	fbAchse_Buerste_030801.IsReset:= P_ServiceAchsen.xStopAktiv_Reset[AxId_Buerste_030801];
	fbAchse_Buerste_030801.IsFreigabe:= P_ServiceAchsen.xFreigabe_Aktiv[AxId_Buerste_030801];
	fbAchse_Buerste_030801.IwZielSollwert:= P_ServiceAchsen.rZielSollwert[AxId_Buerste_030801];
	fbAchse_Buerste_030801.IwSpeed:= P_ServiceAchsen.uiSpeed[AxId_Buerste_030801];
ELSE
	IF	fbEins[iEins_Id].OsAutomatikEin
		OR	fbEins[iEins_Id].OsHandEin
			AND	astrGButtonManTransporte[ID_Buerste_030801_Positionieren].bSchalt
	THEN
		arGZielAchse[AxId_Buerste_030801]:= st_Achse_Buerste_030801.rZiel;
		arGSpeedAchse[AxId_Buerste_030801]:= st_Achse_Buerste_030801.rSpeed;
		abGStartAchse[AxId_Buerste_030801]:= st_Achse_Buerste_030801.xStartPosi;
		abGEichenAchse[AxId_Buerste_030801]:= st_Achse_Buerste_030801.xStartEichen;
		abGFreigabeAchse[AxId_Buerste_030801]:= st_Achse_Buerste_030801.xFreigabe;
	ELSE
		abGStartAchse[AxId_Buerste_030801]:= FALSE;
		abGEichenAchse[AxId_Buerste_030801]:= FALSE;
		abGFreigabeAchse[AxId_Buerste_030801]:= FALSE;
	END_IF;

	fbAchse_Buerste_030801.IsReset:=
		( astrGButtonManTransporte[ID_Buerste_030801_Tippen].bSchalt
			OR	astrGButtonManTransporte[ID_Buerste_030801_Positionieren].bSchalt )
		AND 	strGLmHand.bI_Reset
		OR NOT fbEins[iEins_Id].OsAutomatikEin
			AND	GDat.TrE_Daten[TrEId_030801_Buerste].iReset <> 0;

	fbAchse_Buerste_030801.IsFreigabe:=
		( abGFreigabeAchse[AxId_Buerste_030801]
			AND NOT bFehlerFahrenFreigabe_Buerste_030801
			AND NOT bFehlerFahrenPlus_Buerste_030801
			AND NOT bFehlerFahrenMinus_Buerste_030801
			OR NOT fbAchse_Buerste_030801.IsAutomatik
				AND	fbAchse_Buerste_030801.IsHand )
		AND	fbEins[iEins_Id].OsNotHaltIstOk
		AND NOT fbAchse_Buerste_030801.OwOut.xAchseFehler
		AND	gxAlleTuerenGeschlossen_HardwareC[giSicher_C2_2]
		AND	gxAlleTuerenGeschlossenVerriegelt_HardwareC[giSicher_C2_2]
		AND	gxAlleTuerenGeschlossen_FreigabeAchseC[giSicher_C2_2];

	IF	fbEins[iEins_Id].OsAutomatikEin
		AND	arGSpeedAchse[AxId_Buerste_030801] > 0
	THEN
		fbAchse_Buerste_030801.IwSpeed:=
			LIMIT ( 0.1,arGSpeedAchse[AxId_Buerste_030801],100 );
	ELSE
		fbAchse_Buerste_030801.IwSpeed:= 100;
	END_IF;

	IF	fbAchse_Buerste_030801.IsSichereGeschwindigkeit
	THEN
		fbAchse_Buerste_030801.IwSpeed_HandSlow:= 50;
		fbAchse_Buerste_030801.IwSpeed_HandFast:= 100;
	ELSE
		fbAchse_Buerste_030801.IwSpeed_HandSlow:= 50;
		fbAchse_Buerste_030801.IwSpeed_HandFast:= 100;
	END_IF;

	fbAchse_Buerste_030801.IwBeschleunigung:= st_Achse_Buerste_030801.rBeschleunigung;
	fbAchse_Buerste_030801.IwVerzoegerung:= st_Achse_Buerste_030801.rVerzoegerung;
	fbAchse_Buerste_030801.IwRuck:= st_Achse_Buerste_030801.rRuck;

	fbAchse_Buerste_030801.IsStartEichen:=
		abGEichenAchse[AxId_Buerste_030801]
		AND NOT gxTestbetriebOhneMaschineAktiv;

	fbAchse_Buerste_030801.IwZielSollwert:=
		arGZielAchse[AxId_Buerste_030801];

	fbAchse_Buerste_030801.IsStartAufPosition:=
		abGStartAchse[AxId_Buerste_030801]
		AND 	fbAchse_Buerste_030801.IsFreigabe
		AND	fbAchse_Buerste_030801.OwOut.xAchseGeeicht;

	fbAchse_Buerste_030801.IsNeueGeschwindigkeit:= st_Achse_Buerste_030801.xStartNeueGeschwindigkeit;

	fbAchse_Buerste_030801.IsSonderGeschwindigkeit:= st_Achse_Buerste_030801.xSonderGeschwindigkeit;
	fbAchse_Buerste_030801.IwSonderGeschwindigkeit:= LREAL_TO_REAL ( st_Achse_Buerste_030801.lrSonderGeschwindigkeit );

	fbAchse_Buerste_030801.IsStartNeuesZielWaehrendPosi:= st_Achse_Buerste_030801.xStartNeuesZielWaehrendPosi;
	fbAchse_Buerste_030801.IwNeuesZielWaehrendPosi:= st_Achse_Buerste_030801.rNeuesZielWaehrendPosi;

	IF	fbAchse_Buerste_030801.xZielUmschiessen
	THEN
		st_Achse_Buerste_030801.xStartNeuesZielWaehrendPosi:= FALSE;
	END_IF;

	IF	fbAchse_Buerste_030801.xGeschwindigkeitUmschiessen
	THEN
		st_Achse_Buerste_030801.xStartNeueGeschwindigkeit:= FALSE;
	END_IF;
END_IF;

fbAchse_Buerste_030801();

IF	fbAchse_Buerste_030801.IsHand
	AND	fbAchse_Buerste_030801.IsReset
	OR NOT bAchseBeiStartGeeicht_Buerste_030801
THEN
	abGAchseNeuEichen[AxId_Buerste_030801]:= TRUE;
	bAchseBeiStartGeeicht_Buerste_030801:= TRUE;
END_IF;

(*------------------------------------------------------*)
(*  Handling: -> Jobverteiler                      	  *)
(*------------------------------------------------------*)

st_Achse_Buerste_030801.iID:= AxId_Buerste_030801;
st_Achse_Buerste_030801.xNichtEichen:= TRUE;
st_Achse_Buerste_030801.stVonAchse:= fbAchse_Buerste_030801.OwOut;
st_Achse_Buerste_030801.stVonAchse.xAchseGeeicht:=
	fbAchse_Buerste_030801.OwOut.xAchseGeeicht;

st_Achse_Buerste_030801.xBereit_FuerFahrjob:=
	fbAchse_Buerste_030801.OwOut.xAchseBereit
	AND NOT fbAchse_Buerste_030801.OwOut.xAchseFehler;



(*-----------------------------------------------------------------*)
(* Die globale Struktur für die Leuchtmelde Handtasten beschreiben *)
(*-----------------------------------------------------------------*)
IF	fbAchse_Buerste_030801.IsHand
	AND	astrGButtonManTransporte[ID_Buerste_030801_Tippen].bSchalt
THEN
	IF NOT fbAchse_Buerste_030801.IsEsEndlagePlus
	THEN
		strGLmHand.bQ_Heben:= TRUE;
	END_IF;

	IF NOT fbAchse_Buerste_030801.IsEsEndlageMinus
	THEN
		strGLmHand.bQ_Senken:= TRUE;
	END_IF;
END_IF;



				(*---------------------------------------------------*)
				(*---------------------------------------------------*)
				(*           Freigabe Hardwaren / Software           *)
				(*---------------------------------------------------*)
				(*---------------------------------------------------*)

abGAchseDisable[AxId_Buerste_030801]:=
	GKoAnB[usiBuerste1].xInAktiv;

IF ( fbAchse_Buerste_030801.IsEsEndlageMinus
		OR 	fbAchse_Buerste_030801.IsEsEndlagePlus )
	AND NOT gxTestbetriebOhneMaschineAktiv
THEN
	abGEndlageAngefahren[AxId_Buerste_030801]:= TRUE;
END_IF;

IF	strGLmHand.bI_QuittStoerung
		AND NOT fbAchse_Buerste_030801.IsEsEndlageMinus
		AND NOT fbAchse_Buerste_030801.IsEsEndlagePlus
	OR NOT fbEins[iEins_Id].OsSteuerspannungIstEin
THEN
	abGEndlageFreifahren[AxId_Buerste_030801]:= FALSE;
	abGEndlageAngefahren[AxId_Buerste_030801]:= FALSE;
END_IF;

abGEndlageFreifahren[AxId_Buerste_030801]:=
	fbEins[iEins_Id].OsHandEin
	AND	abGEndlageAngefahren[AxId_Buerste_030801];

aTonGReglerfreigabe[AxId_Buerste_030801].IN:=
	( NOT abGEndlageAngefahren[AxId_Buerste_030801]
		OR	abGEndlageFreifahren[AxId_Buerste_030801] )
	AND	bFreigabeFahren_Buerste_030801
	AND NOT abGAchseDisable[AxId_Buerste_030801]
	AND NOT AxFrNcFehler[AxId_Buerste_030801]
	AND NOT fbAchse_Buerste_030801.OsMFehlerMcBausteine
	AND NOT GKoAnB[usiBuerste1].xInAktiv;

aTonGReglerfreigabe[AxId_Buerste_030801](PT:= T#500MS);

abGReglerfreigabe[AxId_Buerste_030801]:=
	aTonGReglerfreigabe[AxId_Buerste_030801].Q
	OR	aTofGReglerfreigabe_Aus[AxId_Buerste_030801].Q
		AND	AxFrNcFahrePlus[AxId_Buerste_030801]
		AND NOT abGEndlageAngefahren[AxId_Buerste_030801]
	OR	aTofGReglerfreigabe_Aus[AxId_Buerste_030801].Q
		AND	AxFrNcFahreMinus[AxId_Buerste_030801]
		AND NOT abGEndlageAngefahren[AxId_Buerste_030801];

(* Ausschaltverzoegerung Reglerfreigabe *)
aTofGReglerfreigabe_Aus[AxId_Buerste_030801].IN:=
	aTonGReglerfreigabe[AxId_Buerste_030801].IN
		AND  	aTonGReglerfreigabe[AxId_Buerste_030801].Q;
aTofGReglerfreigabe_Aus[AxId_Buerste_030801](PT:= GKoAll.tBisReglerfreigabeAus_BeiNotHalt);

aTonGVorschubfreigabe[AxId_Buerste_030801](PT:= T#500MS);

aTonGVorschubfreigabe[AxId_Buerste_030801].IN:=
	abGReglerfreigabe[AxId_Buerste_030801];

abGVorschubfreigabe[AxId_Buerste_030801]:= aTonGVorschubfreigabe[AxId_Buerste_030801].Q;

abGVorschubfreigabePlus[AxId_Buerste_030801]:=
	NOT fbAchse_Buerste_030801.IsEsEndlagePlus
	OR	gxTestbetriebOhneMaschineAktiv;

abGVorschubfreigabeMinus[AxId_Buerste_030801]:=
	NOT fbAchse_Buerste_030801.IsEsEndlageMinus
	OR	gxTestbetriebOhneMaschineAktiv;

(*---------------------------------------------------*)
(* Achse: Freigabe Software              		     *)
(*---------------------------------------------------*)

AxToNcRfg[AxId_Buerste_030801]:=
	abGReglerfreigabe[AxId_Buerste_030801]
		AND NOT abGAchseDisable[AxId_Buerste_030801];

AxToNcVfp[AxId_Buerste_030801]:=
	abGVorschubfreigabe[AxId_Buerste_030801]
		AND	abGVorschubfreigabePlus[AxId_Buerste_030801]
		AND	aTonGReglerfreigabe[AxId_Buerste_030801].Q
		AND NOT abGAchseDisable[AxId_Buerste_030801];

AxToNcVfm[AxId_Buerste_030801]:=
	abGVorschubfreigabe[AxId_Buerste_030801]
		AND	abGVorschubfreigabeMinus[AxId_Buerste_030801]
		AND	aTonGReglerfreigabe[AxId_Buerste_030801].Q
		AND NOT abGAchseDisable[AxId_Buerste_030801];

(*---------------------------------------------------*)
(* Achse: Ausgänge an Systemmanager schreiben	     *)
(*---------------------------------------------------*)
bQW10SchwertbObZMinus		:= bIW10DirectionMinus;
bQW10SchwertbObZPlus		:= bIW10DirectionPlus;
bQW10SchwertbObZSchnell		:= bIW10VeloHigh;
END_ACTION

ACTION Up_15_EilSchl_PosiBuerste_030801:
(*------------------------------------------------*)
(*------------------------------------------------*)
(* Achse: Jobhandling Positionierung		  *)
(*------------------------------------------------*)
(*------------------------------------------------*)
(*
IF GDat.TrE_Daten[TrEId_030801].iAnzahlPlatten > 0
THEN
	bKleinteilBuerste_030801:= FALSE;

	FOR i:= 1 TO LIMIT(1,GDat.TrE_Daten[TrEId_030801].iAnzahlPlatten,giMaxAnzahlPlattenProSpur)
	DO
		IF	(GDat.TrE_Daten[TrEId_030801].arLaenge[i] <= GKoAnB[usiBuerste1].rMinLaenge_Buerste
				OR GDat.TrE_Daten[TrEId_030801].arBreite[i] <= GKoAnB[usiBuerste1].rMinBreite_Buerste)
		THEN
			bKleinteilBuerste_030801:= TRUE;
			EXIT;
		END_IF;
	END_FOR;

	rDickeBuerste	:= GDat.TrE_Daten[TrEId_030801].arDicke[1];
	rBreiteBuerste	:= GDat.TrE_Daten[TrEId_030801].arBreite[1];

ELSIF ( GDat.TrE_Daten[TrEId_030801].iJobStatus = iDatenAktiv
		OR GDat.TrE_Daten[TrEId_030801].iJobStatus = iUebernahmeGestartet )
	AND GDat.TrE_Daten[TrEId_030801].iAnzahlPlatten = 0
THEN
	bKleinteilBuerste_030801:= FALSE;

	FOR i:= 1 TO LIMIT(1,fbJobBahn030801.strBahnjob_Aktiv.iAnzahlPlatten,giMaxAnzahlPlattenProSpur)
	DO
		IF	(fbJobBahn030801.strBahnjob_Aktiv.arLaenge[i] <= GKoAnB[usiBuerste1].rMinLaenge_Buerste
				OR fbJobBahn030801.strBahnjob_Aktiv.arBreite[i] <= GKoAnB[usiBuerste1].rMinBreite_Buerste)
		THEN
			bKleinteilBuerste_030801:= TRUE;
			EXIT;
		END_IF;
	END_FOR;

	rDickeBuerste	:= fbJobBahn030801.strBahnjob_Aktiv.arDicke[1];
	rBreiteBuerste	:= fbJobBahn030801.strBahnjob_Aktiv.arBreite[1];

ELSIF GDat.TrE_Daten[TrEId_030801].iJobStatus = iSekNichtAktiv
	AND GDat.TrE_Daten[TrEId_030801].iAnzahlPlatten = 0
	AND GDat.TrE_Daten[TrEId_070402].iAnzahlPlatten > 0
THEN

	bKleinteilBuerste_030801:= FALSE;

	FOR i:= 1 TO LIMIT(1,GDat.TrE_Daten[TrEId_070402].iAnzahlPlatten,giMaxAnzahlPlattenProSpur)
	DO
		IF	(GDat.TrE_Daten[TrEId_070402].arLaenge[i] <= GKoAnB[usiBuerste1].rMinLaenge_Buerste
				OR GDat.TrE_Daten[TrEId_070402].arBreite[i] <= GKoAnB[usiBuerste1].rMinBreite_Buerste)
		THEN
			bKleinteilBuerste_030801:= TRUE;
			EXIT;
		END_IF;
	END_FOR;

	rDickeBuerste	:= GDat.TrE_Daten[TrEId_070402].arDicke[1];
	rBreiteBuerste	:= GDat.TrE_Daten[TrEId_070402].arBreite[1];

ELSIF GDat.TrE_Daten[TrEId_030801].iAnzahlPlatten = 0
	AND	GDat.TrE_Daten[TrEId_030801].asBarcode[1] = ''
	AND 	strGHdshk_Bahn030801.str_BahnStatus = iAutomatikBereitJob
	AND NOT strGHdshk_Bahn030801.b_BahnBelegt
THEN
	bKleinteilBuerste_030801:= FALSE;
END_IF;

fbTOF_BuersteAntriebEin_030801(
		IN:= strGHdshk_Bahn030801.b_BahnVor,
		PT:= t#5s,
		Q=> ,
		ET=> );

fbEntprellenHoehenkontrolle_030801(
	IsSensor:= NOT bIW308Hoehenkontr
					AND FALSE,
	tEntprell_Belegt:= t#1s,
	tEntprell_Frei:= t#1s,
	OsSensor=> );

IF	fbEntprellenHoehenkontrolle_030801.OsSensor
	AND NOT gxTestbetriebOhneMaschineAktiv
THEN
	bQ_MFehlerHoehenkontrolle030801:= TRUE;

ELSIF	bQ_MFehlerHoehenkontrolle030801
	AND (strGLmHand.bI_QuittStoerung
		OR (NOT fbEntprellenHoehenkontrolle_030801.OsSensor
			AND AxFrNc_fPosIst[AxId_Buerste_030801] >= (GDat.TrE_Daten[TrEId_030801].arDicke[1] - fbBuerste_030801.rToleranzBuerste)))
THEN
	bQ_MFehlerHoehenkontrolle030801:= FALSE;
END_IF
*)

fbBuerste_030801(
	sI_Name							:= '03.08.01_Buerste',
	uiI_AxId_Oben					:= AxId_Buerste_030801,
	uiI_ProId						:= P_BahnJob,
	bI_Hand							:= fbEins[iEins_Id].OsHandEin,
	bI_Automatik					:= fbEins[iEins_Id].OsAutomatikEin,
	bI_Reset						:= strGLmHand.bI_Reset
								 	 	AND ( astrGButtonManTransporte[ID_Buerste_030801_Tippen].bSchalt
									 		 OR	astrGButtonManTransporte[ID_Buerste_030801_Positionieren].bSchalt ),
	bI_QuittStoerung				:= strGLmHand.bI_QuittStoerung
										OR fbEins[iEins_Id].OsImpulsSteuerspannungEin,
	bI_ZyklusBeenden				:= fbEins[iEins_Id].OsZyklusBeenden
										OR	Aufruf_Allgemein.bAnforderungAnlageAus,
	bI_StoerungBuerstenAntriebOben	:= NOT bIW10SchwertbuersteObBtp,
	bI_StoerungBuerstenAntriebUnten	:= NOT bIW10SchwertbuersteUntBtp,
	bI_StoerungAchse				:= FALSE,
	bI_SicherheitOK					:= gxSicherheitsBereichQuittiertC[giSicher_C2_2],
	bI_Kleinteile					:= bKleinteilBuerste_030801,
	bI_BuersteZu					:= TRUE,
	bI_BuersteAntriebEin			:= strGHdshk_Bahn030801.b_BahnVor,
	bI_TeileBuersten				:= TRUE,
	bI_TeileReinigen				:= fbTOF_BuersteAntriebEin_030801.Q,
	bI_IngromatEin					:= FALSE,
	bI_FahrtInGrundOhneEichen		:= astrGButtonManTransporte[ID_Buerste_030801_Tippen].bSchalt
										OR	astrGButtonManTransporte[ID_Buerste_030801_Positionieren].bSchalt,
	bI_FreigabeAufPosition			:= fbBuerste_030801.rI_Dicke > 0,
	bI_EichenManuell				:= TRUE,
	bI_Testbetrieb					:= gxTestbetriebOhneMaschineAktiv,
	bI_ImpulsInit					:= bGImpulsInitSprache,
	rI_Dicke						:= fbJobBahn030801.strBahnjob_Aktiv.arDicke[1],
	rI_Breite						:= fbJobBahn030801.strBahnjob_Aktiv.arBreite[1], 
	strI_Para						:= GKoAnB[usiBuerste1],
	strIO_TrE_Extern 				:= GDat.TrE_Daten[TrEId_030801_Buerste],
	strIO_Hubachse_Oben				:= st_Achse_Buerste_030801,
	abQ_Blasventil					=> ,
	bQ_BuersteOeffnen				=> ,
	bQ_BuersteObenEin				=> bQW10SchwertbuersteObEin,
	bQ_BuersteUntenEin				=> bQW10SchwertbuersteUntEin,
	bQ_Reinigen						=> bQW10SchwertbReinigEin,
	bQ_Ingromat						=> ,
	bQ_ZyklusBeendet				=> ,
	bQ_Grundstellung				=> ,
	bQ_SchleichenEichenOben			=> ,
	bQ_IstwertSetzenOben=> ,
	bQ_MStoerungBuerstenAntriebOben=> ,
	bQ_MStoerungBuerstenAntriebUnten=> ,
	uiQ_Ablaufstatus=> , 
	strQ_Status=> );

	
IF	astrGButtonManTransporte[ID_Buerste_030801_Tippen].bSchalt
	OR	astrGButtonManTransporte[ID_Buerste_030801_Positionieren].bSchalt
THEN
	TZeile.Aktiv := TRUE;
	TZeile.Wert  := REAL_TO_INT(AxFrNc_fPosIst[AxId_Buerste_030801]);
END_IF;

IF	( fbBuerste_030801.strQ_Status = iAutomatikBereitJob
		AND	fbBuerste_030801.rI_Dicke > 0
		AND	st_Achse_Buerste_030801.xBereit_FuerFahrjob
		AND 	(( ABS (( fbBuerste_030801.rI_Dicke + fbBuerste_030801.strI_Para.rOeffnungswertKleinteile_Oben ) - fbBuerste_030801.rIstwert ) <= fbBuerste_030801.rToleranzBuerste
				AND	fbBuerste_030801.bI_Kleinteile )
			OR	( ABS ( fbBuerste_030801.rI_Dicke - fbBuerste_030801.rIstwert ) <= fbBuerste_030801.rToleranzBuerste
				AND NOT fbBuerste_030801.bI_Kleinteile )))
	OR	fbBuerste_030801.strI_Para.xInAktiv
THEN
	bBuersteInPostion_030801:= TRUE;
ELSE
	bBuersteInPostion_030801:= FALSE;
END_IF;
END_ACTION

ACTION Up_16_Anschlag_030201:

fbAnschlag_030201(
	IsHand									:= fbEins[iEins_Id].OsHandEin
												OR ( NOT fbEins[iEins_Id].OsAutomatikEin
													AND ( GDat.TrE_Daten[TrEId_030201_Roll1].iReset <> 0
														OR	GDat.TrE_Daten[TrEId_030202_Roll2].iReset <> 0 ) ),
	IsAutomatik								:= fbEins[iEins_Id].OsAutomatikEin,
	IsReset									:= astrGButtonManTransporte[ID_Anschlag030201].bSchalt
												AND	strGLmHand.bI_Reset
												OR ( NOT fbEins[iEins_Id].OsAutomatikEin
													AND ( GDat.TrE_Daten[TrEId_030201_Roll1].iReset <> 0
														OR GDat.TrE_Daten[TrEId_030202_Roll2].iReset <> 0 )),
	IsQuittStoerung							:= strGLmHand.bI_QuittStoerung,
	IsTestbetrieb							:= gxTestbetriebOhneMaschineAktiv,
	IsNotHaltIstOK							:= TRUE,
	IsFreigabe_Automatik					:= TRUE,
	IsStoerungAntrieb						:= strGStoerungen[iEins_Id].bStoerungDruckluft,
	IsSicherheitOK							:= gxSicherheitsBereichQuittiertC[giSicher_C2_1],
	IsTHandVor								:= astrGButtonManTransporte[ID_Anschlag030201].bSchalt
												AND	strGLmHand.bI_Senken,
	IsTHandZurueck							:= astrGButtonManTransporte[ID_Anschlag030201].bSchalt
												AND	strGLmHand.bI_Heben,
	IsDauerlauf_Aktivieren					:= astrGButtonManTransporte[ID_Anschlag030201].bSchalt
												AND	gxDauerlauf_Aktiv,
	IsHand_Takt								:= gTakt22,
	IsGrundstellung							:= bIW302Anschlag1Sek1GS
												AND NOT gxTestbetriebOhneMaschineAktiv
												OR	gxTestbetriebOhneMaschineAktiv
													AND	fbAnschlag_030201.OsGrundstellung,
	IsArbeitsstellung						:= bIW302Anschlag1Sek1AS
												AND NOT gxTestbetriebOhneMaschineAktiv
												OR	gxTestbetriebOhneMaschineAktiv
													AND	fbAnschlag_030201.OsArbeitsstellung,
	IwMode									:= 3,
	IwMode_NotHalt							:= 0,
	IwDoJob									:= strGHdshk_Anschlag030201.str_DoJob,
	IsFreigabeGrundposition					:= TRUE,
	IsGrundpositionArbeitsstellung			:= strGHdshk_Anschlag030201.b_Arbeitsstellung,
	IsKeineGrundposition					:= FALSE,
	IsOhneUeberwachung						:= FALSE,
	IsGesetzterOutMerken					:= TRUE,
	IsClearOut_NachJob						:= FALSE,
	IsOutAnlassen_Hand						:= TRUE,
	IsOutAnlassen_Stoerung					:= TRUE,
	IsPositionsUeberwachung					:= TRUE,
	IsBewegungsUeberwachung					:= TRUE,
	IwBisGrundstellung						:= strGHdshk_Anschlag030201.tBisGrundstellung,
	IwBisArbeitsstellung					:= strGHdshk_Anschlag030201.tBisArbeitsstellung,
	IwMaxLaufzeitZylinder					:= strGHdshk_Anschlag030201.tMaxLaufzeit,
	IwBisDrucklos							:= strGHdshk_Anschlag030201.tBisDrucklos,
	OsGrundstellung							=> bQW302AnschlagSek1GS,
	OsArbeitsstellung						=> bQW302AnschlagSek1AS,
	OwJobAktiv								=> strGHdshk_Anschlag030201.str_JobAktiv,
	OwStatus								=> strGHdshk_Anschlag030201.str_ZylinderStatus,
	OwAblaufStatus							=> strGHdshk_Anschlag030201.i_AblaufStatus,
	OsMStoerungAntrieb						=> strGHdshk_Anschlag030201.b_MStoerungAntrieb,
	OsMMaxLaufzeit_Ein						=> strGHdshk_Anschlag030201.b_MMaxLaufzeit_Ein,
	OsMMaxLaufzeit_Aus						=> strGHdshk_Anschlag030201.b_MMaxLaufzeit_Aus,
	OsMPositionsUeberwachung_Ein			=> strGHdshk_Anschlag030201.b_MPositionsUeberwachung_Ein,
	OsMPositionsUeberwachung_Aus			=> strGHdshk_Anschlag030201.b_MPositionsUeberwachung_Aus,
	OsMBewegungsUeberwachung				=> strGHdshk_Anschlag030201.b_MBewegungsUeberwachung);

	
strGHdshk_Anschlag030201.b_Arbeitsstellung:= fbAnschlag_030201.IsArbeitsstellung;
strGHdshk_Anschlag030201.b_Grundstellung:= fbAnschlag_030201.IsGrundstellung;

(* Jobstatus setzen *)

IF	strGHdshk_Anschlag030201.str_DoJob > eJob_KeinJob
	AND	strGHdshk_Anschlag030201.str_DoJob = strGHdshk_Anschlag030201.str_JobAktiv
	OR	fbAnschlag_030201.IsHand
		AND fbAnschlag_030201.IsReset
THEN
	strGHdshk_Anschlag030201.str_DoJob:= eJob_KeinJob;
END_IF;

(* Handbetrieb *)

IF	fbAnschlag_030201.IsHand
	AND	astrGButtonManTransporte[ID_Anschlag030201].bSchalt
THEN
	IF NOT fbAnschlag_030201.IsArbeitsstellung
	THEN
		strGLmHand.bQ_Senken:= TRUE;
	END_IF;

	IF NOT fbAnschlag_030201.IsGrundstellung
	THEN
		strGLmHand.bQ_Heben:= TRUE;
	END_IF;
END_IF;

(* Meldungen *)

fbMeldungenAnschlag_030201(
	uiI_FehlerId			:= 3000,
	strIO_GHdshk_Zylinder	:= strGHdshk_Anschlag030201,
	strIO_Stoerungen		:= strGStoerungen[iEins_Id]);


(* Ansteuerung Automatik *)

IF	strGHdshk_Anschlag030201 .str_DoJob = eJob_KeinJob
	AND	strGHdshk_Anschlag030201.str_JobAktiv = eJob_KeinJob
	AND	strGHdshk_Anschlag030201.str_ZylinderStatus = iAutomatikBereitJob
THEN
	IF  GDat.TrE_Daten[TrEId_030301].iJobStatus = iDatenAktiv
		AND	fbJobBahn030301.strBahnjob_Aktiv.diZielId = strGHdshk_Bahn030301.di_PlatzId
		AND	fbJobBahn030301.strBahnjob_Aktiv.diQuellId = strGHdshk_Bahn030201_Roll1.di_PlatzId
		AND	strGHdshk_Bahn030201_Roll1.str_JobAktiv_AufBahn = eRolljobKeinJob
		AND strGHdshk_Bahn030201_Roll1.str_JobAktiv_VonBahn = eRolljobKeinJob
		AND	strGHdshk_Bahn030202_Roll2.str_JobAktiv_AufBahn = eRolljobKeinJob
		AND strGHdshk_Bahn030202_Roll2.str_JobAktiv_VonBahn = eRolljobKeinJob
		OR ( GDat.TrE_Daten[TrEId_030201_Roll1].iJobStatus = iDatenAktiv				(* Ein Job nach dem anderen *)
			AND NOT strGHdshk_Bahn030201_Roll1.b_BahnBelegt
			AND NOT strGHdshk_Bahn030202_Roll2.b_BahnBelegt
			AND GDat.TrE_Daten[TrEId_030201_Roll1].iAnzahlPlatten = 0
			AND GDat.TrE_Daten[TrEId_030202_Roll2].iAnzahlPlatten = 0
			AND	strGHdshk_Bahn030201_Roll1.i_BahnV2_AufBahn_BereitFuerJob = 0
			AND strGHdshk_Bahn030201_Roll1.i_BahnV2_VonBahn_BereitFuerJob = 0			
			AND	strGHdshk_Bahn030202_Roll2.i_BahnV2_AufBahn_BereitFuerJob = 0
			AND strGHdshk_Bahn030202_Roll2.i_BahnV2_VonBahn_BereitFuerJob = 0 )
		AND NOT strGHdshk_Anschlag030201.b_Grundstellung
	THEN
		strGHdshk_Anschlag030201.str_DoJob:= eJob_Grundstellung;

	ELSIF (( GDat.TrE_Daten[TrEId_030201_Roll1].iJobStatus = iDatenAktiv				(* Ein Job nach dem anderen *)
			AND	fbJobBahn030201.strBahnjob_Aktiv_Sek_1.diZielId = strGHdshk_Bahn030201_Roll1.di_PlatzId
			AND	fbJobBahn030201.strBahnjob_Aktiv_Sek_1.diQuellId = strGHdshk_Bahn030101.di_PlatzId
			AND NOT strGHdshk_Bahn030201_Roll1.b_BahnBelegt
			AND strGHdshk_Bahn030202_Roll2.b_BahnBelegt
			AND GDat.TrE_Daten[TrEId_030201_Roll1].iAnzahlPlatten = 0
			AND GDat.TrE_Daten[TrEId_030202_Roll2].iAnzahlPlatten <> 0
			AND	strGHdshk_Bahn030201_Roll1.i_BahnV2_AufBahn_BereitFuerJob = 0
			AND strGHdshk_Bahn030201_Roll1.i_BahnV2_VonBahn_BereitFuerJob = 0 )
		OR (strGHdshk_Bahn030201_Roll1.str_JobAktiv_AufBahn = eRolljobAufBahnPosiVorlauf		(* Ein Job mit vollständigem Bild *)	
			AND	strGHdshk_Bahn030202_Roll2.str_JobAktiv_AufBahn = eRolljobAufBahnPosiVorlauf
			AND GDat.TrE_Daten[TrEId_030201_Roll1].iAnzahlPlatten <> 0
			AND GDat.TrE_Daten[TrEId_030202_Roll2].iAnzahlPlatten <> 0
			AND strGHdshk_Bahn030202_Roll2.str_PlattenPos.arPlattenPos[1] >= strGHdshk_Bahn030202_Roll2.str_Bahndaten.rGesamtLaenge - 400 ))
		AND NOT strGHdshk_Anschlag030201.b_Arbeitsstellung
	THEN
		strGHdshk_Anschlag030201.str_DoJob:= eJob_Arbeitsstellung;
	END_IF;
END_IF;
END_ACTION

ACTION Up_19_Bahn_040101_Extern:
IF	fbJobBahn040101.bQ_GrundOK
THEN
	strGHdshk_BahnExternW2.str_BahnStatus:= GDat.TrE_Daten[TrEId_ExternW2].iAktivStatus;
ELSE
	strGHdshk_BahnExternW2.str_BahnStatus:= iAutomatikBereitJob;
END_IF;


IF	fbJobBahn040101.bKeinJobInJobzeile
	AND	fbJobBahn040101.iAnzahlJobsAktiv = 0
	AND	fbJobBahn040101.bQ_GrundOK
	AND NOT fbJobBahn040101.bQ_ResetAktiv
	AND	bFreigabeFuerJob_C2_2
	AND	GDat.TrE_Daten[TrEId_ExternW2].iJobStatus = iSekNichtAktiv
	AND	strGADSKomEmpfangVonPos0400.strJob_Daten.iJobStatus = iJobzeileAktiv
	AND	strGADSKomEmpfangVonPos0400.strJob_Daten.diQuellId = strGHdshk_Bahn030801.di_PlatzId
	AND	strGADSKomEmpfangVonPos0400.strJob_Daten.diZielId = strGHdshk_BahnExternW2.di_PlatzId
	AND	strGADSKomEmpfangVonPos0400.strJob_Daten.iAnzahlPlatten > 0
	AND	diJobIdAltExternW2 <> strGADSKomEmpfangVonPos0400.strJob_Daten.diJobID
	AND ( strGADSKomEmpfangVonPos0400.strTrE_Daten.iJobStatus = iDatenAktiv
		OR	strGADSKomEmpfangVonPos0400.strTrE_Daten.iJobStatus = iUebernahmeGestartet )
THEN
		fbJobDaten_In_ZielTrE(
			iMode_Copy			:= 3,
			iMode_Daten			:= 0,
			iBarcodePruefen		:= 0,
			Jobzeile			:= strGADSKomEmpfangVonPos0400.strJob_Daten,
			TrE_Daten			:= TrE_DatenJobExternW2 );

		fbQuellTrE_In_JobDaten(
			bI_JobSofortBeenden	:= FALSE,
			iI_AnzahlPlatten		:= TrE_DatenJobExternW2.iAnzahlPlatten,
			diI_QuellId			:= strGHdshk_Bahn030801.di_PlatzId,
			diI_ZielId			:= strGHdshk_BahnExternW2.di_PlatzId,
			strIO_TrE_Quelle		:= TrE_DatenJobExternW2,
			strIO_ArbTab_Job_Ziel	:= GJobDat.ArbTab_Job[TrEId_ExternW2] );

		diJobIdAltExternW2:= strGADSKomEmpfangVonPos0400.strJob_Daten.diJobID;
ELSE
		fbTrE_Daten_Leer(TrE_Daten:= TrE_DatenJobExternW2 );
END_IF;


IF	( GDat.TrE_Daten[TrEId_ExternW2].iJobStatus = iDatenAktiv
		OR GDat.TrE_Daten[TrEId_ExternW2].iJobStatus = iUebernahmeGestartet )
	AND	strGADSKomEmpfangVonPos0400.strJob_Daten.iJobStatus <> iJobzeileAktiv
	OR	GDat.TrE_Daten[TrEId_030801].iReset <> 0
THEN
	GDat.TrE_Daten[TrEId_ExternW2].iReset:= 1;
END_IF;



fbJobBahn040101(
	bI_MitPCJob                               := NOT gxTestbetriebOhnePCJobs,
	bI_FreigabeJobErzeugenSPS_Vorg            := gxTestbetriebOhnePCJobs,
	bI_FreigabeJobErzeugenSPS_Nachf           := FALSE,
	bI_FreigabeResetJob                       := astrGButtonManTransporte[ID_Bahn030801].bSchalt,
	bI_FreigabeResetBahn                      := astrGButtonManTransporte[ID_Bahn030801].bSchalt,
	bI_FreigabeFuerJob                        := bFreigabeFuerJob_C2_2,
	bI_ZusatzFreigabe                         := TRUE,
	bI_FreigabeFuerBuchen                     := bFreigabeFuerBuchen_C2_2,
	bI_MitAufBahnBeiVonBahn                   := FALSE,
	bI_Querfoerderer                          := FALSE,
	bI_FreigabeAnBahnanfang                   := FALSE,
	bI_FreigabeAnsBahnende                    := FALSE,
	bI_ScannenAktiv                           := FALSE,
	bI_Testbetrieb                            := gxTestbetriebOhneMaschineAktiv,
	bI_FehlerQuittScanner                     := FALSE,
	bI_BeiResetJoblisteLoeschen               := NOT bG3TecIstLeitsystem,
	iI_MaxAnzahlJobs                          := 1,
	iI_MaxAnzahlNoRead                        := 1,
	uiI_ProId                                 := P_BahnJob,
	diI_SperrenQuellBahnNrVonPortal           := 0,
	diI_SperrenZielBahnNrVonPortal            := 0,
	tI_BisScannerDatenDa                      := t#0s,
	tI_Systemzeit                             := P_SystemzeitAuswerten.tDatumZeit_PC,
	strIO_GHdshk                              := strGHdshk_BahnExternW2,
	strIO_GHdshk_Vorg                         := strGHdshk_Bahn030801,
	strIO_GHdshk_Nachf                        := strBahnaustausch_Leer,
	strIO_TrE                                 := GDat.TrE_Daten[TrEId_ExternW2],
	strIO_TrE_Vorg                            := GDat.TrE_Daten[TrEId_030801],
	strIO_TrE_Nachf                           := TrE_Daten_Leer,
	strIO_ArbTab_Job                          := GJobDat.ArbTab_Job[TrEId_ExternW2],
	strIO_GLmHand                             := strGLmHand,
	fbIO_Scanner                              := fbScanner_Leer,
	bQ_GrundOK                                => ,
	bQ_ResetAktiv                             => ,
	bQ_ScannerHatNichtGelesen                 => ,
	bQ_ScannerFalscherBarcode                 => ,
	bQ_ScannerMaxAnzahlNoRead                 => );


FOR i:= 0 TO giListenLaenge_Job
DO
	IF	GJobDat.ArbTab_Job[TrEId_ExternW2].JobZeile[i].iJobStatus = iJobzeileBeendet
	THEN
		GJobDat.ArbTab_Job[TrEId_ExternW2].JobZeile[i].iJobStatus:= iJobzeileGeloescht;
	END_IF
END_FOR;
END_ACTION

ACTION Up_21_Bahn_030801:

fbHardwareBahn030801(
	uiI_ProId									:= P_BahnHardware,
	uiI_TrEId									:= TrEId_030801,
	uiI_AxId									:= 0,
	uiI_FehlerId								:= 4650,
	sI_Bahnname									:= '03.08.01',
	bI_Hand										:= fbEins[iEins_Id].OsHandEin,
	bI_Automatik								:= fbEins[iEins_Id].OsAutomatikEin,
	bI_Testbetrieb								:= gxTestbetriebOhneMaschineAktiv,
	bI_SicherheitOK								:= gxSicherheitsBereichQuittiertC[giSicher_C2_2],
	bI_FreigabeAutomatik						:= TRUE,
	bI_FreigabeHandVorZurueck					:= astrGButtonManTransporte[ID_Bahn030801].bSchalt,
	bI_BahnDarfZurueckHand						:= FALSE,
	bI_FreigabeReset							:= astrGButtonManTransporte[ID_Bahn030801].bSchalt,
	bI_StoerungAntrieb							:= NOT fbG6UmrichterBahn030801.bQ_Betriebsbereit
													OR NOT fbG6UmrichterBahn030802.bQ_Betriebsbereit,
	bI_Anfang									:= NOT bIW308Transp1Anf,
	bI_BelegtKontrolle							:= FALSE,
	bI_Ende										:= NOT bIW308Transp2End,
	bI_VorZurueckInversHand						:= FALSE,
	bI_AbbruchPosi_AufBahn						:= FALSE,
	bI_AbbruchPosi_VonBahn						:= FALSE,
	bI_BahnenGrundSchnell						:= FALSE,
	bI_GrundZurueck								:= FALSE,
	bI_OhneSynchronVonBahn						:= FALSE,
	bI_NachlaufAmAnfangEnde						:= FALSE,
	bI_MitUeberwachungTeilNichtFreigegeben		:= FALSE,
	bI_ImpulsInit								:= bGImpulsInitSprache,
	bI_OhneImpulsgeber							:= FALSE,
	bI_AutoHandaufgabeAktiv						:= FALSE,
	bI_AutoHandentnahmeAktiv					:= FALSE,
	strIO_GHdshk								:= strGHdshk_Bahn030801,
	strIO_GHdshk_Vorg							:= strGHdshk_Bahn030701_Roll,
	strIO_GHdshk_Nachf							:= strGHdshk_BahnExternW2,
	strIO_GLmHand								:= strGLmHand,
	strIO_TrE									:= GDat.TrE_Daten[TrEId_030801],
	strIO_Stoerungen							:= strGStoerungen[iEins_Id]);

fbG6UmrichterBahn030801(
	sI_NetIDMaster						:= P_Ueberwachung_EtherCat.sNetId,
	sI_PfadXML							:= sGG6XMLPfad,
	sI_PfadSonderDatensatz				:= '',
	sI_Name								:= '=W308.EA1+S1-TA1',
	uiI_FxId							:= FxId_030801,
	uiI_ProId							:= P_Umrichter,
	uiI_DevID							:= uiIDevID,
	diI_Statuswort						:= udiIW308TA1Statuswort,
	usiI_Umrichterstatus				:= usiIW308TA1UmrichterStatus,
	uiI_Datensatz						:= 1,
	iI_Istfrequenz						:= uiIW308TA1Istfrequenz,
	tI_ZeitBremse						:= t#500ms,
	rI_Beschleunigung					:= 0.1,
	rI_Verzoegerung						:= 0.1,
	rI_Sollgeschwindigkeit				:= LREAL_TO_REAL(ABS(strGHdshk_Bahn030801.lr_Bahnspeed_Vorgabe)),
	rI_Maxgeschwindigkeit				:= strGHdshk_Bahn030801.str_BahnSpeed.rVmaxSpeed,
	bI_Aktiv							:= TRUE,
	bI_FehlerQuitt						:= strGLmHand.bI_QuittStoerung,
	bI_Testbetrieb						:= gxTestbetriebOhneMaschineAktiv,
	bI_StartUmrichter					:= gxSicherheitsBereichQuittiertC[giSicher_C2_2],
	bI_Reglerfreigabe					:= gxSicherheitsBereichVerzOKC[giSicher_C2_2],
	bI_DrehrichtungVor					:= strGHdshk_Bahn030801.b_BahnVor,
	bI_DrehrichtungZurueck				:= strGHdshk_Bahn030801.b_BahnZurueck,
	bI_EtherCATOK						:= P_Ueberwachung_EtherCat.xAlles_OK,
	bI_DrehInv							:= TRUE,
	uiQ_EtherCATAdresse					=> uiGEtherCATAdresse_KEB[FxId_030801],
	iQ_Sollwert							=> uiQW308TA1Sollw,
	lrQ_Istwert							=> strGHdshk_Bahn030801.lr_Bahnspeed_Ist,
	diQ_Control							=> udiQW308TA1Control,
	bQ_Betriebsbereit					=> ,
	bQ_BremseLoesen						=> ,
	bQ_FehlerKEBDatenDownload			=> ,
	bQ_FehlerKeinIMAUmrichter			=> ,
	bQ_FehlerXMLDatei					=> ,
	bQ_FehlerParaLesen					=> ,
	bQ_FehlerParaSchreiben				=> ,
	bQ_FehlerAdresseLesen				=> ,
	strQ_Umrichterstatus				=> );

Aufruf_DisplayKEB.arI_DisplayKEB[FxId_030801]:=
	fbG6UmrichterBahn030801.strQ_Umrichterstatus.sConverterState;

fbG6UmrichterBahn030802(
	sI_NetIDMaster						:= P_Ueberwachung_EtherCat.sNetId,
	sI_PfadXML							:= sGG6XMLPfad,
	sI_PfadSonderDatensatz				:= '',
	sI_Name								:= '=W308.EA2+S1-TA1',
	uiI_FxId							:= FxId_030802,
	uiI_ProId							:= P_Umrichter,
	uiI_DevID							:= uiIDevID,
	diI_Statuswort						:= udiIW308TA2Statuswort,
	usiI_Umrichterstatus				:= usiIW308TA2UmrichterStatus,
	uiI_Datensatz						:= 1,
	iI_Istfrequenz						:= uiIW308TA2Istfrequenz,
	tI_ZeitBremse						:= t#500ms,
	rI_Beschleunigung					:= 0.1,
	rI_Verzoegerung						:= 0.1,
	rI_Sollgeschwindigkeit				:= LREAL_TO_REAL(ABS(strGHdshk_Bahn030801.lr_Bahnspeed_Vorgabe)),
	rI_Maxgeschwindigkeit				:= strGHdshk_Bahn030801.str_BahnSpeed.rVmaxSpeed,
	bI_Aktiv							:= TRUE,
	bI_FehlerQuitt						:= strGLmHand.bI_QuittStoerung,
	bI_Testbetrieb						:= gxTestbetriebOhneMaschineAktiv,
	bI_StartUmrichter					:= gxSicherheitsBereichQuittiertC[giSicher_C2_2],
	bI_Reglerfreigabe					:= gxSicherheitsBereichVerzOKC[giSicher_C2_2],
	bI_DrehrichtungVor					:= strGHdshk_Bahn030801.b_BahnVor,
	bI_DrehrichtungZurueck				:= strGHdshk_Bahn030801.b_BahnZurueck,
	bI_EtherCATOK						:= P_Ueberwachung_EtherCat.xAlles_OK,
	bI_DrehInv							:= TRUE,
	uiQ_EtherCATAdresse					=> uiGEtherCATAdresse_KEB[FxId_030802],
	iQ_Sollwert							=> uiQW308TA2Sollw,
	lrQ_Istwert							=> strGHdshk_Bahn030801.lr_Bahnspeed_Ist,
	diQ_Control							=> udiQW308TA2Control,
	bQ_Betriebsbereit					=> ,
	bQ_BremseLoesen						=> ,
	bQ_FehlerKEBDatenDownload			=> ,
	bQ_FehlerKeinIMAUmrichter			=> ,
	bQ_FehlerXMLDatei					=> ,
	bQ_FehlerParaLesen					=> ,
	bQ_FehlerParaSchreiben				=> ,
	bQ_FehlerAdresseLesen				=> ,
	strQ_Umrichterstatus				=> );

Aufruf_DisplayKEB.arI_DisplayKEB[FxId_030802]:=
	fbG6UmrichterBahn030802.strQ_Umrichterstatus.sConverterState;
	
	
fbJobBahn030801(
	bI_MitPCJob								:= TRUE,
	bI_FreigabeJobErzeugenSPS_Vorg			:= FALSE,
	bI_FreigabeJobErzeugenSPS_Nachf			:= FALSE,
	bI_FreigabeResetJob						:= astrGButtonManTransporte[ID_Bahn030801].bSchalt,
	bI_FreigabeResetBahn					:= astrGButtonManTransporte[ID_Bahn030801].bSchalt,
	bI_FreigabeFuerJob						:= bFreigabeFuerJob_C2_2,
	bI_ZusatzFreigabe                         := GDat.TrE_Daten[TrEId_030801].iJobStatus = iDatenAktiv
												AND fbBuerste_030801.strQ_Status = iAutomatikBereitJob
												AND	fbBuerste_030801.bQ_Grundstellung
												AND ( ABS(fbBuerste_030801.rQ_Plattendicke - fbJobBahn030801.strBahnjob_Aktiv.arDicke[1]) <= fbBuerste_030801.rToleranzBuerste
														 OR REAL_TO_INT(fbAchse_Buerste_030801.rAxFrNc_fPosIst) >=  fbJobBahn030801.strBahnjob_Aktiv.arDicke[1]
															AND fbJobBahn030801.strBahnjob_Aktiv.arDicke[1] <= 13  )
												AND fbBuerste_030801.rQ_Plattendicke > 0
												AND NOT strGHdshk_Bahn030801.b_BahnBelegt
												OR	GKoAnB[usiBuerste1].xInAktiv,
	bI_FreigabeFuerBuchen					:= bFreigabeFuerBuchen_C2_2,
	bI_MitAufBahnBeiVonBahn					:= FALSE,
	bI_BilderSammeln						:= FALSE, 
	bI_Querfoerderer						:= FALSE,
	bI_FreigabeAnBahnanfang					:= FALSE,
	bI_FreigabeAnsBahnende					:= FALSE,
	bI_ScannenAktiv							:= FALSE,
	bI_Testbetrieb							:= gxTestbetriebOhneMaschineAktiv,
	bI_FehlerQuittScanner					:= FALSE,
	bI_BeiResetJoblisteLoeschen				:= NOT bG3TecIstLeitsystem,
	iI_MaxAnzahlJobs						:= 1,
	iI_MaxAnzahlNoRead						:= 1,
	uiI_ProId								:= P_BahnJob,
	diI_SperrenQuellBahnNrVonPortal			:= 0,
	diI_SperrenZielBahnNrVonPortal			:= 0,
	tI_BisScannerDatenDa					:= t#0s,
	tI_Systemzeit							:= P_SystemzeitAuswerten.tDatumZeit_PC,
	strIO_GHdshk							:= strGHdshk_Bahn030801,
	strIO_GHdshk_Vorg						:= strGHdshk_Bahn030701_Roll,
	strIO_GHdshk_Nachf						:= strGHdshk_BahnExternW2,
	strIO_TrE								:= GDat.TrE_Daten[TrEId_030801],
	strIO_TrE_Vorg							:= GDat.TrE_Daten[TrEId_030701],
	strIO_TrE_Nachf							:= GDat.TrE_Daten[TrEId_ExternW2],
	strIO_ArbTab_Job						:= GJobDat.ArbTab_Job[TrEId_030801],
	strIO_GLmHand							:= strGLmHand,
	fbIO_Scanner							:= fbScanner_Leer,
	bQ_GrundOK								=> ,
	bQ_ResetAktiv							=> ,
	bQ_ScannerHatNichtGelesen				=> ,
	bQ_ScannerFalscherBarcode				=> ,
	bQ_ScannerMaxAnzahlNoRead				=> );
END_ACTION

ACTION Up_22_Bahn_030701:
fbHardwareBahn030701(
			uiI_ProId:= P_BahnHardware,
			uiI_TrEId:= TrEId_030701,
			uiI_AxId_Roll1:= 0,
			uiI_AxId_Riem1:= 0,
			uiI_AxId_Riem2:= 0,
			uiI_FehlerId_Roll1:= 4500,
			uiI_FehlerId_Riem1:= 4550,
			uiI_FehlerId_Riem2:= 5600,
			sI_Bahnname:= '03.07.01',
			bI_Hand:= fbEins[iEins_Id].OsHandEin,
			bI_Automatik:= fbEins[iEins_Id].OsAutomatikEin,
			bI_Testbetrieb:= gxTestbetriebOhneMaschineAktiv,
			bI_SicherheitOK:= gxSicherheitsBereichQuittiertC[giSicher_C2_1],
			bI_FreigabeAutomatik:= TRUE,
			bI_FreigabeHandVorZurueck_Roll1:= astrGButtonManTransporte[ID_Bahn030701_Roll].bSchalt,
			bI_FreigabeHandVorZurueck_Riem1:= astrGButtonManTransporte[ID_Bahn030702_Riem1].bSchalt,
			bI_FreigabeHandVorZurueck_Riem2:= astrGButtonManTransporte[ID_Bahn030703_Riem2].bSchalt,
			bI_BahnDarfZurueckHand_Roll1:= FALSE,
			bI_BahnDarfZurueckHand_Riem1:= TRUE,
			bI_BahnDarfZurueckHand_Riem2:= TRUE,
			bI_FreigabeHandHebenSenkenSek1:= astrGButtonManTransporte[ID_Bahn030702_Riem1].bSchalt
									OR astrGButtonManTransporte[ID_Bahn030701_Roll].bSchalt,
			bI_FreigabeHandHebenSenkenSek2:= astrGButtonManTransporte[ID_Bahn030703_Riem2].bSchalt
									OR astrGButtonManTransporte[ID_Bahn030701_Roll].bSchalt,
			bI_FreigabeReset:= astrGButtonManTransporte[ID_Bahn030701_Roll].bSchalt
									OR astrGButtonManTransporte[ID_Bahn030702_Riem1].bSchalt
									OR astrGButtonManTransporte[ID_Bahn030703_Riem2].bSchalt,
			bI_StoerungAntrieb_Roll1:=NOT fbG6UmrichterBahn030701_Roll.bQ_Betriebsbereit ,
			bI_Anfang_Roll1:= NOT bIW307Transp11TeilVorAnschl OR NOT bIW307Transp12TeilVorAnschl,
			bI_Ende_Roll1:= NOT bIW308Transp1Anf,
			bI_AufFoerderhoehe_Roll1:= bIW307Transp2GS,
			bI_StoerungAntrieb_Riem1:= NOT fbG6UmrichterBahn030702_Riem1.bQ_Betriebsbereit,
			bI_Anfang_Riem1:= NOT bIW307Transp11Anf,
			bI_Ende_Riem1:= NOT bIW307Transp11TeilVorAnschl
								AND strGHdshk_Bahn030702_Riem1.r_PosiRestwert_AufBahn = 0,
			bI_AufFoerderhoehe_Riem1:= bIW307Transp2AS,
			bI_StoerungAntrieb_Riem2:= NOT fbG6UmrichterBahn030703_Riem2.bQ_Betriebsbereit,
			bI_Anfang_Riem2:= NOT bIW307Transp12Anf,
			bI_Ende_Riem2:= NOT bIW307Transp12TeilVorAnschl
								AND strGHdshk_Bahn030703_Riem2.r_PosiRestwert_AufBahn = 0,
			bI_AufFoerderhoehe_Riem2:= bIW307Transp2AS,
			bI_HebenSenkenInvers:= FALSE,
			bI_VorZurueckInversHand:= FALSE,
			bI_AbbruchPosi_AufBahn_Roll1:= FALSE,
			bI_AbbruchPosi_AufBahn_Riem1:= FALSE,
			bI_AbbruchPosi_AufBahn_Riem2:= FALSE,
			bI_AbbruchPosi_VonBahn_Roll1:= FALSE,
			bI_AbbruchPosi_VonBahn_Riem1:= FALSE,
			bI_AbbruchPosi_VonBahn_Riem2:= FALSE,
			bI_BahnenGrundSchnell_Sek_1:= FALSE,
			bI_BahnenGrundSchnell_Sek_2:= FALSE,
			bI_HubGrundWennFrei_Sek_1:= FALSE,
			bI_HubGrundWennFrei_Sek_2:= FALSE,
			bI_HubArbeitWennFrei_Sek_1:= FALSE,
			bI_HubArbeitWennFrei_Sek_2:= FALSE,
			bI_HubGrundWennBelegt_Sek_1:= FALSE,
			bI_HubGrundWennBelegt_Sek_2:= FALSE,
			bI_HubArbeitWennBelegt_Sek_1:= FALSE ,
			bI_HubArbeitWennBelegt_Sek_2:= FALSE ,
			bI_OhneSynchronVonBahn_Roll1:= FALSE,
			bI_OhneSynchronVonBahn_Riem1:= FALSE,
			bI_OhneSynchronVonBahn_Riem2:= FALSE,
			bI_VorgRiemHatNurEineSpur:= TRUE,
			bI_NachfRiemHatNurEineSpur:= FALSE,
			bI_MitUeberwachungTeilNichtFreigegeben:= FALSE,
			bI_ImpulsInit:= bGImpulsInitSprache,
			bI_OhneImpulsgeber_Roll1:= FALSE,
			bI_OhneImpulsgeber_Riem1:= FALSE,
			bI_OhneImpulsgeber_Riem2:= FALSE,
			strIO_GHdshk_Roll1:= strGHdshk_Bahn030701_Roll,
			strIO_GHdshk_Roll1_Vorg:= strBahnaustausch_Leer,
			strIO_GHdshk_Roll1_Nachf:= strGHdshk_Bahn030801,
			strIO_GHdshk_Riem1:= strGHdshk_Bahn030702_Riem1,
			strIO_GHdshk_Riem1_Vorg:= strGHdshk_Bahn030601,
			strIO_GHdshk_Riem1_Nachf:= strBahnaustausch_Leer,
			strIO_GHdshk_Riem2:=  strGHdshk_Bahn030703_Riem2,
			strIO_GHdshk_Riem2_Vorg:= strGHdshk_Bahn030601,
			strIO_GHdshk_Riem2_Nachf:= strBahnaustausch_Leer,
			strIO_GLmHand:= strGLmHand,
			strIO_TrE:= GDat.TrE_Daten[TrEId_030701],
			strIO_Stoerungen:=  strGStoerungen[iEins_Id],
			bQ_Sektion1AS=> bQW307Transp2AS,
			bQ_Sektion1GS=> bQW307Transp2GS,
			bQ_Sektion2AS=> bQW307Transp2AS,
			bQ_Sektion2GS=> bQW307Transp2GS );

fbG6UmrichterBahn030701_Roll(
			sI_NetIDMaster					:= P_Ueberwachung_EtherCat.sNetId,
			sI_PfadXML						:= sGG6XMLPfad,
			sI_PfadSonderDatensatz			:= '',
			sI_Name							:= '=W307.EA1+S1-TA1',
			uiI_DevID						:= uiIDevID,
			uiI_FxId						:= FxId_030701_Roll,
			uiI_ProId						:= P_Umrichter,
			diI_Statuswort					:= udiIW307TA1Statuswort,
			usiI_Umrichterstatus			:= usiIW307TA1UmrichterStatus,
			uiI_Datensatz					:= 1,
			iI_Istfrequenz					:= uiIW307TA1Istfrequenz,
			tI_ZeitBremse					:= t#500ms,
			rI_Beschleunigung				:= 0.1,
			rI_Verzoegerung					:= 0.1,
			rI_Sollgeschwindigkeit			:= ABS(strGHdshk_Bahn030701_Roll.lr_Bahnspeed_Vorgabe),
			rI_Maxgeschwindigkeit			:= strGHdshk_Bahn030701_Roll.str_BahnSpeed.rVmaxSpeed,
			bI_Aktiv						:= TRUE,
			bI_FehlerQuitt					:= strGLmHand.bI_QuittStoerung,
			bI_Testbetrieb					:= gxTestbetriebOhneMaschineAktiv,
			bI_StartUmrichter				:= gxSicherheitsBereichQuittiertC[giSicher_C2_1],
			bI_Reglerfreigabe				:= gxSicherheitsBereichVerzOKC[giSicher_C2_1],
			bI_DrehrichtungVor				:= strGHdshk_Bahn030701_Roll.b_BahnVor,
			bI_DrehrichtungZurueck			:= strGHdshk_Bahn030701_Roll.b_BahnZurueck,
			bI_EtherCATOK					:= P_Ueberwachung_EtherCat.xAlles_OK,
			bI_DrehInv						:= TRUE,
			uiQ_EtherCATAdresse			    => uiGEtherCATAdresse_KEB[FxId_030701_Roll],
			iQ_Sollwert						=> uiQW307TA1Sollw,
			lrQ_Istwert						=> strGHdshk_Bahn030701_Roll.lr_Bahnspeed_Ist,
			diQ_Control						=> udiQW307TA1Control,
			bQ_Betriebsbereit				=> ,
			bQ_BremseLoesen					=> bQW307Bremse1Loe,
			bQ_FehlerKEBDatenDownload		=> ,
			bQ_FehlerKeinIMAUmrichter		=> ,
			bQ_FehlerXMLDatei				=> ,
			bQ_FehlerParaLesen				=> ,
			bQ_FehlerParaSchreiben			=> ,
			bQ_FehlerAdresseLesen			=> ,
			strQ_Umrichterstatus			=> );

Aufruf_DisplayKEB.arI_DisplayKEB[FxId_030701_Roll]:=
			fbG6UmrichterBahn030701_Roll.strQ_Umrichterstatus.sConverterState;

fbG6UmrichterBahn030702_Riem1(
		sI_NetIDMaster					:= P_Ueberwachung_EtherCat.sNetId,
		sI_PfadXML						:= sGG6XMLPfad,
		sI_PfadSonderDatensatz			:= '',
		sI_Name							:= '=W307.EB11+S1-TA1',
		uiI_DevID						:= uiIDevID,
		uiI_FxId						:= FxId_030702_Riem1,
		uiI_ProId						:= P_Umrichter,
		diI_Statuswort					:= udiIW307TA11Statuswort,
		usiI_Umrichterstatus			:= usiIW307TA11UmrichterStatus,
		uiI_Datensatz					:= 1,
		iI_Istfrequenz					:= uiIW307TA11Istfrequenz,
		tI_ZeitBremse					:= t#500ms,
		rI_Beschleunigung				:= 0.1,
		rI_Verzoegerung					:= 0.1,
		rI_Sollgeschwindigkeit			:= ABS(strGHdshk_Bahn030702_Riem1.lr_Bahnspeed_Vorgabe),
		rI_Maxgeschwindigkeit			:= strGHdshk_Bahn030702_Riem1.str_BahnSpeed.rVmaxSpeed,
		bI_Aktiv						:= TRUE,
		bI_FehlerQuitt					:= strGLmHand.bI_QuittStoerung,
		bI_Testbetrieb					:= gxTestbetriebOhneMaschineAktiv,
		bI_StartUmrichter					:= gxSicherheitsBereichQuittiertC[giSicher_C2_1],
		bI_Reglerfreigabe					:= gxSicherheitsBereichVerzOKC[giSicher_C2_1],
		bI_DrehrichtungVor				:= strGHdshk_Bahn030702_Riem1.b_BahnVor,
		bI_DrehrichtungZurueck				:= strGHdshk_Bahn030702_Riem1.b_BahnZurueck,
		bI_EtherCATOK					:= P_Ueberwachung_EtherCat.xAlles_OK,
		bI_DrehInv						:= FALSE,//TRUE,
		uiQ_EtherCATAdresse			    	=> uiGEtherCATAdresse_KEB[FxId_030702_Riem1],
		iQ_Sollwert						=> uiQW307TA11Sollw,
		lrQ_Istwert						=> strGHdshk_Bahn030702_Riem1.lr_Bahnspeed_Ist,
		diQ_Control						=> udiQW307TA11Control,
		bQ_Betriebsbereit					=> ,
		bQ_BremseLoesen					=> ,
		bQ_FehlerKEBDatenDownload			=> ,
		bQ_FehlerKeinIMAUmrichter			=> ,
		bQ_FehlerXMLDatei					=> ,
		bQ_FehlerParaLesen				=> ,
		bQ_FehlerParaSchreiben				=> ,
		bQ_FehlerAdresseLesen				=> ,
		strQ_Umrichterstatus				=> );

Aufruf_DisplayKEB.arI_DisplayKEB[FxId_030702_Riem1]:=
		fbG6UmrichterBahn030702_Riem1.strQ_Umrichterstatus.sConverterState;


fbG6UmrichterBahn030703_Riem2(
		sI_NetIDMaster					:= P_Ueberwachung_EtherCat.sNetId,
		sI_PfadXML						:= sGG6XMLPfad,
		sI_PfadSonderDatensatz			:= '',
		sI_Name							:= '=W307.EB12+S1-TA1',
		uiI_DevID						:= uiIDevID,
		uiI_FxId						:= FxId_030703_Riem2,
		uiI_ProId						:= P_Umrichter,
		diI_Statuswort					:= udiIW307TA12Statuswort,
		usiI_Umrichterstatus			:= usiIW307TA12UmrichterStatus,
		uiI_Datensatz					:= 1,
		iI_Istfrequenz					:= uiIW307TA12Istfrequenz,
		tI_ZeitBremse					:= t#500ms,
		rI_Beschleunigung				:= 0.1,
		rI_Verzoegerung					:= 0.1,
		rI_Sollgeschwindigkeit			:= ABS(strGHdshk_Bahn030703_Riem2.lr_Bahnspeed_Vorgabe),
		rI_Maxgeschwindigkeit			:= strGHdshk_Bahn030703_Riem2.str_BahnSpeed.rVmaxSpeed,
		bI_Aktiv						:= TRUE,
		bI_FehlerQuitt					:= strGLmHand.bI_QuittStoerung,
		bI_Testbetrieb					:= gxTestbetriebOhneMaschineAktiv,
		bI_StartUmrichter				:= gxSicherheitsBereichQuittiertC[giSicher_C2_1],
		bI_Reglerfreigabe				:= gxSicherheitsBereichVerzOKC[giSicher_C2_1],
		bI_DrehrichtungVor				:= strGHdshk_Bahn030703_Riem2.b_BahnVor,
		bI_DrehrichtungZurueck			:= strGHdshk_Bahn030703_Riem2.b_BahnZurueck,
		bI_EtherCATOK					:= P_Ueberwachung_EtherCat.xAlles_OK,
		bI_DrehInv						:= FALSE,
		uiQ_EtherCATAdresse			    => uiGEtherCATAdresse_KEB[FxId_030703_Riem2],
		iQ_Sollwert						=> uiQW307TA12Sollw,
		lrQ_Istwert						=> strGHdshk_Bahn030703_Riem2.lr_Bahnspeed_Ist,
		diQ_Control						=> udiQW307TA12Control,
		bQ_Betriebsbereit				=> ,
		bQ_BremseLoesen					=> ,
		bQ_FehlerKEBDatenDownload		=> ,
		bQ_FehlerKeinIMAUmrichter		=> ,
		bQ_FehlerXMLDatei				=> ,
		bQ_FehlerParaLesen				=> ,
		bQ_FehlerParaSchreiben			=> ,
		bQ_FehlerAdresseLesen			=> ,
		strQ_Umrichterstatus			=> );

Aufruf_DisplayKEB.arI_DisplayKEB[FxId_030703_Riem2]:=
		fbG6UmrichterBahn030703_Riem2.strQ_Umrichterstatus.sConverterState;

fbJobBahn030701(
		bI_MitPCJob								:= TRUE,
		bI_FreigabeJobErzeugenSPS_Roll1_Vorg	:= FALSE,
		bI_FreigabeJobErzeugenSPS_Roll1_Nachf	:= FALSE,
		bI_FreigabeJobErzeugenSPS_Riem1_Vorg	:= FALSE,
		bI_FreigabeJobErzeugenSPS_Riem1_Nachf	:= FALSE,
		bI_FreigabeJobErzeugenSPS_Riem2_Vorg	:= FALSE,
		bI_FreigabeJobErzeugenSPS_Riem2_Nachf	:= FALSE,
		bI_FreigabeResetJob						:= astrGButtonManTransporte[ID_Bahn030701_Roll].bSchalt
													OR astrGButtonManTransporte[ID_Bahn030702_Riem1].bSchalt
													OR astrGButtonManTransporte[ID_Bahn030703_Riem2].bSchalt,
		bI_FreigabeResetBahn					:= astrGButtonManTransporte[ID_Bahn030701_Roll].bSchalt
													OR astrGButtonManTransporte[ID_Bahn030702_Riem1].bSchalt
													OR astrGButtonManTransporte[ID_Bahn030703_Riem2].bSchalt,
		bI_FreigabeFuerJob					:= bFreigabeFuerJob_C2_1,
		bI_ZusatzFreigabe					:= TRUE,
		bI_FreigabeFuerBuchen				:= bFreigabeFuerBuchen_C2_1,
		bI_MitAufBahnBeiVonBahn				:= FALSE,
		bI_Querfoerderer_Roll				:= FALSE,
		bI_Querfoerderer_Riem				:= TRUE,
		bI_FreigabeAnBahnanfang_Roll1		:= FALSE,
		bI_FreigabeAnsBahnende_Roll1		:= FALSE,
		bI_FreigabeAnBahnanfang_Riem1		:= FALSE,
		bI_FreigabeAnsBahnende_Riem1		:= FALSE,
		bI_FreigabeAnBahnanfang_Riem2		:= FALSE,
		bI_FreigabeAnsBahnende_Riem2		:= FALSE,
		bI_VorgRiemHatNurEineSpur			:= TRUE,
		bI_NachfRiemHatNurEineSpur			:= FALSE,
		bI_BahnHKStop_Roll1					:= FALSE,
		bI_BahnHKStop_Riem1					:= FALSE,
		bI_BahnHKStop_Riem2					:= FALSE,
		bI_ScannenAktiv_Roll1				:= FALSE,
		bI_ScannenAktiv_Riem1				:= FALSE,
		bI_ScannenAktiv_Riem2				:= FALSE,
		bI_Testbetrieb						:= gxTestbetriebOhneMaschineAktiv,
		bI_FehlerQuittScanner_Roll1			:= FALSE,
		bI_FehlerQuittScanner_Riem1			:= FALSE,
		bI_FehlerQuittScanner_Riem2			:= FALSE,
		bI_BeiResetJoblisteLoeschen			:= NOT bG3TecIstLeitsystem,
		iI_MaxAnzahlJobs					:= 1,
		iI_MaxAnzahlNoRead					:= 1,
		uiI_ProId							:= P_BahnJob,
	(*	diI_SperrenQuellBahnNrVonPortal:= ,
		diI_SperrenZielBahnNrVonPortal:= , *)
		tI_BisScannerDatenDa				:= t#0s,
		tI_Systemzeit						:= P_SystemzeitAuswerten.tDatumZeit_PC,
		strIO_GHdshk_Roll1					:= strGHdshk_Bahn030701_Roll,
		strIO_GHdshk_Roll1_Vorg				:= strBahnaustausch_Leer,
		strIO_GHdshk_Roll1_Nachf			:= strGHdshk_Bahn030801,
		strIO_GHdshk_Riem1					:= strGHdshk_Bahn030702_Riem1,
		strIO_GHdshk_Riem1_Vorg				:= strGHdshk_Bahn030601,
		strIO_GHdshk_Riem1_Nachf			:= strBahnaustausch_Leer,
		strIO_GHdshk_Riem2					:= strGHdshk_Bahn030703_Riem2,
		strIO_GHdshk_Riem2_Vorg				:= strGHdshk_Bahn030601,
		strIO_GHdshk_Riem2_Nachf			:= strBahnaustausch_Leer,
		strIO_TrE							:= GDat.TrE_Daten[TrEId_030701],
		strIO_TrE_Roll1_Vorg				:= TrE_Daten_Leer,
		strIO_TrE_Roll1_Nachf				:= GDat.TrE_Daten[TrEId_030801],
		strIO_TrE_Riem1_Vorg				:= GDat.TrE_Daten[TrEId_030601],
		strIO_TrE_Riem1_Nachf				:= TrE_Daten_Leer,
		strIO_TrE_Riem2_Vorg				:= GDat.TrE_Daten[TrEId_030601],
		strIO_TrE_Riem2_Nachf				:= TrE_Daten_Leer,
		strIO_ArbTab_Job					:= GJobDat.ArbTab_Job[TrEId_030701],
		strIO_ArbTab_Job_Riem1_Vorg			:= GJobDat.ArbTab_Job[TrEId_030601],
		strIO_ArbTab_Job_Riem2_Vorg			:= GJobDat.ArbTab_Job[TrEId_030601],
		strIO_ArbTab_Job_Riem1_Nachf		:= strArbTab_Job_Leer,
		strIO_ArbTab_Job_Riem2_Nachf		:= strArbTab_Job_Leer,
		strIO_GLmHand						:= strGLmHand,
		fbIO_Scanner_Roll1					:= fbScanner_Leer,
		fbIO_Scanner_Riem1					:= fbScanner_Leer,
		fbIO_Scanner_Riem2					:= fbScanner_Leer,
		bQ_GrundOK							=> ,
		bQ_ResetAktiv						=> ,
		bQ_ScannerHatNichtGelesen_Roll1		=> ,
		bQ_ScannerHatNichtGelesen_Riem1		=> ,
		bQ_ScannerHatNichtGelesen_Riem2		=> ,
		bQ_ScannerFalscherBarcode_Roll1		=> ,
		bQ_ScannerFalscherBarcode_Riem1		=> ,
		bQ_ScannerFalscherBarcode_Riem2		=> ,
		bQ_ScannerMaxAnzahlNoRead_Roll1		=> ,
		bQ_ScannerMaxAnzahlNoRead_Riem1		=> ,
		bQ_ScannerMaxAnzahlNoRead_Riem2		=> );
END_ACTION

ACTION Up_23_Bahn_030601:
(*--------------------------*)
(* Sollposition Wippe       *)
(*--------------------------*)

IF	GDat.TrE_Daten[TrEId_030601].iJobStatus = iDatenAktiv
    	AND GDat.TrE_Daten[TrEId_030601].iAnzahlPlatten <= 2
THEN
	IF	fbJobBahn030601.strBahnjob_Aktiv.diQuellId = strGHdshk_Bahn030501.di_PlatzId
	THEN
		iWippe_030601_SollAufPos:= 1;

	ELSIF fbJobBahn030601.strBahnjob_Aktiv.diQuellId = strGHdshk_Bahn031501.di_PlatzId
	THEN
		iWippe_030601_SollAufPos:= 2;

	ELSIF fbJobBahn030601.strBahnjob_Aktiv.diQuellId = strGHdshk_Bahn032501.di_PlatzId
	THEN
		iWippe_030601_SollAufPos:= 3;
	END_IF
END_IF;

(*--------------------------*)
(* Zwischenmerker schreiben *)
(*--------------------------*)

IF	iWippe_030601_IstAufPos = 1
THEN
	strGHdshk_Zwischen_030601:= strGHdshk_Bahn030501;
	strTrEDaten_Zwischen_030601:= GDat.TrE_Daten[TrEId_030501];

ELSIF iWippe_030601_IstAufPos = 2
THEN
	strGHdshk_Zwischen_030601:= strGHdshk_Bahn031501;
	strTrEDaten_Zwischen_030601:= GDat.TrE_Daten[TrEId_031501];

ELSIF iWippe_030601_IstAufPos = 3
THEN
	strGHdshk_Zwischen_030601:= strGHdshk_Bahn032501;
	strTrEDaten_Zwischen_030601:= GDat.TrE_Daten[TrEId_032501];
ELSE
	strGHdshk_Zwischen_030601:= strBahnaustausch_Leer;
	strTrEDaten_Zwischen_030601:= TrE_Daten_Leer;
END_IF;

(*----------------------------*)
(* Rampen koppeln zum Sammeln *)
(*----------------------------*)

IF	strGHdshk_Bahn030501.str_DoJob_VonBahn = eRolljobVonBahnPosiVorlauf
	OR	strGHdshk_Bahn030501.str_JobAktiv_VonBahn = eRolljobVonBahnPosiVorlauf
THEN
	strGHdshk_Bahn030601.str_BahnRampen.lrBeschleunigung_mms2:=
		strGHdshk_Bahn030501.str_BahnRampen.lrBeschleunigung_mms2;
		
ELSIF strGHdshk_Bahn031501.str_DoJob_VonBahn = eRolljobVonBahnPosiVorlauf
	OR	strGHdshk_Bahn031501.str_JobAktiv_VonBahn = eRolljobVonBahnPosiVorlauf
THEN
	strGHdshk_Bahn030601.str_BahnRampen.lrBeschleunigung_mms2:=
		strGHdshk_Bahn031501.str_BahnRampen.lrBeschleunigung_mms2;
		
ELSIF strGHdshk_Bahn032501.str_DoJob_VonBahn = eRolljobVonBahnPosiVorlauf
	OR	strGHdshk_Bahn032501.str_JobAktiv_VonBahn = eRolljobVonBahnPosiVorlauf
THEN
	strGHdshk_Bahn030601.str_BahnRampen.lrBeschleunigung_mms2:=
		strGHdshk_Bahn032501.str_BahnRampen.lrBeschleunigung_mms2;
END_IF;



fbHardwareBahn030601(
	uiI_ProId							:= P_BahnHardware,
	uiI_TrEId							:= TrEId_030601,
	uiI_AxId							:= 0,
	uiI_FehlerId						:= 4450,
	sI_Bahnname							:= '03.06.01',
	bI_Hand								:= fbEins[iEins_Id].OsHandEin,
	bI_Automatik						:= fbEins[iEins_Id].OsAutomatikEin,
	bI_Testbetrieb						:= gxTestbetriebOhneMaschineAktiv,
	bI_SicherheitOK						:= gxSicherheitsBereichQuittiertC[giSicher_C2_1],
	bI_FreigabeAutomatik				:= TRUE,
	bI_FreigabeHandVorZurueck			:= astrGButtonManTransporte[ID_Bahn030601].bSchalt,
	bI_BahnDarfZurueckHand				:= TRUE,
	bI_FreigabeReset					:= astrGButtonManTransporte[ID_Bahn030601].bSchalt,
	bI_StoerungAntrieb					:= NOT fbG6UmrichterBahn030601.bQ_Betriebsbereit,
	bI_Anfang							:= ( NOT bIW306Transp1AnfSpur1
												OR NOT bIW306Transp1AnfSpur2 )
											OR strGHdshk_Bahn030501.str_JobAktiv_VonBahn = eRolljobVonBahnPosiVorlauf
												AND ( NOT bIW305Transp1EndSpur1
														OR NOT bIW305Transp1EndSpur2 )
											OR strGHdshk_Bahn031501.str_JobAktiv_VonBahn = eRolljobVonBahnPosiVorlauf
												AND ( NOT bIW315Transp1EndSpur1
														OR NOT bIW315Transp1EndSpur2 )
											OR strGHdshk_Bahn032501.str_JobAktiv_VonBahn = eRolljobVonBahnPosiVorlauf
												AND ( NOT bIW325Transp1EndSpur1
														OR NOT bIW325Transp1EndSpur2 ),
										(*	OR	strGHdshk_Bahn030601.str_JobAktiv_AufBahn = eRolljobAnBahnanfangRuecklauf
												AND NOT strGHdshk_Bahn030601.b_LiEnde, *)
	bI_BelegtKontrolle					:= FALSE,
	bI_Ende								:= NOT bIW307Transp11Anf
												OR NOT bIW307Transp12Anf,//OR bIW307Transp12Anf,
	bI_VorZurueckInversHand				:= FALSE,
	bI_AbbruchPosi_AufBahn				:= FALSE,
	bI_AbbruchPosi_VonBahn				:= FALSE,
	bI_BahnenGrundSchnell				:= FALSE,
	bI_GrundZurueck						:= FALSE,
	bI_OhneSynchronVonBahn				:= FALSE,
	bI_NachlaufAmAnfangEnde				:= FALSE,
	bI_MitUeberwachungTeilNichtFreigegeben		:= FALSE,
	bI_ImpulsInit						:= bGImpulsInitSprache,
	bI_OhneImpulsgeber					:= FALSE,
	bI_AutoHandaufgabeAktiv				:= FALSE,
	bI_AutoHandentnahmeAktiv			:= FALSE,
	strIO_GHdshk						:= strGHdshk_Bahn030601,
	strIO_GHdshk_Vorg					:= strGHdshk_Zwischen_030601,
	strIO_GHdshk_Nachf					:= strGHdshk_Bahn030702_Riem1,
	strIO_GLmHand						:= strGLmHand,
	strIO_TrE							:= GDat.TrE_Daten[TrEId_030601],
	strIO_Stoerungen					:= strGStoerungen[iEins_Id]);

fbG6UmrichterBahn030601(
	sI_NetIDMaster						:= P_Ueberwachung_EtherCat.sNetId,
	sI_PfadXML							:= sGG6XMLPfad,
	sI_PfadSonderDatensatz				:= '',
	sI_Name								:= '=W306.EA1+S1-TA1',
	uiI_FxId							:= FxId_030601,
	uiI_ProId							:= P_Umrichter,
	uiI_DevID							:= uiIDevID,
	diI_Statuswort						:= udiIW306TA1Statuswort,
	usiI_Umrichterstatus				:= usiIW306TA1UmrichterStatus,
	uiI_Datensatz						:= 1,
	iI_Istfrequenz						:= uiIW306TA1Istfrequenz,
	tI_ZeitBremse						:= t#500ms,
	rI_Beschleunigung					:= 0.1,
	rI_Verzoegerung						:= 0.1,
	rI_Sollgeschwindigkeit				:= LREAL_TO_REAL(ABS(strGHdshk_Bahn030601.lr_Bahnspeed_Vorgabe)),
	rI_Maxgeschwindigkeit				:= strGHdshk_Bahn030601.str_BahnSpeed.rVmaxSpeed,
	bI_Aktiv							:= TRUE,
	bI_FehlerQuitt						:= strGLmHand.bI_QuittStoerung,
	bI_Testbetrieb						:= gxTestbetriebOhneMaschineAktiv,
	bI_StartUmrichter					:= gxSicherheitsBereichQuittiertC[giSicher_C2_1],
	bI_Reglerfreigabe					:= gxSicherheitsBereichVerzOKC[giSicher_C2_1],
	bI_DrehrichtungVor					:= strGHdshk_Bahn030601.b_BahnVor,
	bI_DrehrichtungZurueck				:= strGHdshk_Bahn030601.b_BahnZurueck,
	bI_EtherCATOK						:= P_Ueberwachung_EtherCat.xAlles_OK,
	bI_DrehInv							:= FALSE,
	uiQ_EtherCATAdresse					=> uiGEtherCATAdresse_KEB[FxId_030601],
	iQ_Sollwert							=> uiQW306TA1Sollw,
	lrQ_Istwert							=> strGHdshk_Bahn030601.lr_Bahnspeed_Ist,
	diQ_Control							=> udiQW306TA1Control,
	bQ_Betriebsbereit					=> ,
	bQ_BremseLoesen						=> ,
	bQ_FehlerKEBDatenDownload			=> ,
	bQ_FehlerKeinIMAUmrichter			=> ,
	bQ_FehlerXMLDatei					=> ,
	bQ_FehlerParaLesen					=> ,
	bQ_FehlerParaSchreiben				=> ,
	bQ_FehlerAdresseLesen				=> ,
	strQ_Umrichterstatus				=> );


fbJobBahn030601(
	bI_MitPCJob							:= TRUE,
	bI_FreigabeJobErzeugenSPS_Vorg		:= FALSE,
	bI_FreigabeJobErzeugenSPS_Nachf		:= FALSE,
	bI_FreigabeResetJob					:= astrGButtonManTransporte[ID_Bahn030601].bSchalt,
	bI_FreigabeResetBahn				:= astrGButtonManTransporte[ID_Bahn030601].bSchalt,
	bI_FreigabeFuerJob					:= bFreigabeFuerJob_C1_1,
	bI_ZusatzFreigabe					:= GDat.TrE_Daten[TrEId_030601].iJobStatus = iDatenAktiv
											AND  bFreigabeJob_Wippe_030601
											AND ( bSpaltlichschrankenOK_Wippe_030601
												OR	iWippe_030601_IstAufPos = iWippe_030601_SollAufPos )
											AND ( fbJobBahn030601.strBahnjob_Aktiv.diQuellId = strGHdshk_Bahn030501.di_PlatzId
													AND	iWippe_030601_IstAufPos = 1
												OR	fbJobBahn030601.strBahnjob_Aktiv.diQuellId = strGHdshk_Bahn031501.di_PlatzId
													AND	iWippe_030601_IstAufPos = 2
												OR	fbJobBahn030601.strBahnjob_Aktiv.diQuellId = strGHdshk_Bahn032501.di_PlatzId
													AND	iWippe_030601_IstAufPos = 3 )
											AND strGHdshk_Zwischen_030601.di_PlatzId = fbJobBahn030601.strBahnjob_Aktiv.diQuellId,					
	bI_FreigabeFuerBuchen				:= bFreigabeFuerBuchen_C1_1,
	bI_MitAufBahnBeiVonBahn				:= FALSE,
	bI_Querfoerderer					:= FALSE,
	bI_FreigabeAnBahnanfang				:= FALSE,
	bI_FreigabeAnsBahnende				:= FALSE,
	bI_BilderSammeln					:= fbJobBahn030601.strBahnjob_Aktiv.aiPos_X[1] <= 1
											AND	fbJobBahn030601.strBahnjob_Aktiv.aiPos_X[2] <= 1
											AND	fbJobBahn030601.strBahnjob_Aktiv.aiPos_X[3] <= 1
											AND	fbJobBahn030601.strBahnjob_Aktiv.aiPos_X[4] <= 1
											AND	fbJobBahn030601.strBahnjob_Aktiv.arLaenge[1] <= strGHdshk_Bahn030601.str_Bahndaten.rRastermass_Laenge_LaengstePlatte
											AND	fbJobBahn030601.strBahnjob_Aktiv.arLaenge[2] <= strGHdshk_Bahn030601.str_Bahndaten.rRastermass_Laenge_LaengstePlatte ,
	bI_ScannenAktiv						:= FALSE,
	bI_Testbetrieb						:= gxTestbetriebOhneMaschineAktiv,
	bI_FehlerQuittScanner				:= FALSE,
	bI_BeiResetJoblisteLoeschen			:= NOT bG3TecIstLeitsystem,
	iI_MaxAnzahlJobs					:= 1,
	iI_MaxAnzahlNoRead					:= 1,
	uiI_ProId							:= P_BahnJob,
	diI_SperrenQuellBahnNrVonPortal		:= 0,
	diI_SperrenZielBahnNrVonPortal		:= 0,
	tI_BisScannerDatenDa				:= T#0S,
	tI_Systemzeit						:= P_SystemzeitAuswerten.tDatumZeit_PC,
	strIO_GHdshk						:= strGHdshk_Bahn030601,
	strIO_GHdshk_Vorg					:= strGHdshk_Zwischen_030601,
	strIO_GHdshk_Nachf					:= strGHdshk_Bahn030702_Riem1,
	strIO_TrE							:= GDat.TrE_Daten[TrEId_030601],
	strIO_TrE_Vorg						:= strTrEDaten_Zwischen_030601,
	strIO_TrE_Nachf						:= GDat.TrE_Daten[TrEId_030701],
	strIO_ArbTab_Job					:= GJobDat.ArbTab_Job[TrEId_030601],
	strIO_GLmHand						:= strGLmHand,
	fbIO_Scanner						:= fbScanner_Leer,
	bQ_GrundOK							=> ,
	bQ_ResetAktiv						=> ,
	bQ_ScannerHatNichtGelesen			=> ,
	bQ_ScannerFalscherBarcode			=> ,
	bQ_ScannerMaxAnzahlNoRead			=> );

(*---------------------------------*)
(* Zwischenmerker zurueckschreiben *)
(*---------------------------------*)

IF	iWippe_030601_IstAufPos = 1
THEN
	strGHdshk_Bahn030501:= strGHdshk_Zwischen_030601;
	GDat.TrE_Daten[TrEId_030501]:= strTrEDaten_Zwischen_030601;

ELSIF iWippe_030601_IstAufPos = 2
THEN
	strGHdshk_Bahn031501:= strGHdshk_Zwischen_030601;
	GDat.TrE_Daten[TrEId_031501]:= strTrEDaten_Zwischen_030601;

ELSIF iWippe_030601_IstAufPos = 3
THEN
	strGHdshk_Bahn032501:= strGHdshk_Zwischen_030601;
	GDat.TrE_Daten[TrEId_032501]:= strTrEDaten_Zwischen_030601;

END_IF;
END_ACTION

ACTION Up_24_Bahn_032501:
fbHardwareBahn032501(
	uiI_ProId								:= P_BahnHardware,
	uiI_TrEId								:= TrEId_032501,
	uiI_AxId								:= 0,
	uiI_FehlerId							:= 4900,
	sI_Bahnname								:= '03.25.01',
	bI_Hand									:= fbEins[iEins_Id].OsHandEin,
	bI_Automatik							:= fbEins[iEins_Id].OsAutomatikEin,
	bI_Testbetrieb							:= gxTestbetriebOhneMaschineAktiv,
	bI_SicherheitOK							:= gxSicherheitsBereichQuittiertC[giSicher_C2_1],
	bI_FreigabeAutomatik					:= TRUE,
	bI_FreigabeHandVorZurueck				:= astrGButtonManTransporte[ID_Bahn032501].bSchalt,
	bI_BahnDarfZurueckHand					:= TRUE,
	bI_FreigabeReset						:= astrGButtonManTransporte[ID_Bahn032501].bSchalt,
	bI_StoerungAntrieb						:= NOT fbG6UmrichterBahn032501.bQ_Betriebsbereit,
	bI_Anfang								:= NOT bIW325Transp1AnfSpur1
													OR NOT bIW325Transp1AnfSpur2,
	bI_BelegtKontrolle						:= FALSE,
	bI_Ende									:= NOT bIW325Transp1EndSpur1
													OR NOT bIW325Transp1EndSpur2,
	bI_VorZurueckInversHand					:= FALSE,
	bI_AbbruchPosi_AufBahn					:= FALSE,
	bI_AbbruchPosi_VonBahn					:= FALSE,
	bI_BahnenGrundSchnell					:= FALSE,
	bI_GrundZurueck							:= FALSE,
	bI_OhneSynchronVonBahn					:= FALSE,
	bI_NachlaufAmAnfangEnde					:= FALSE,
	bI_MitUeberwachungTeilNichtFreigegeben	:= FALSE,
	bI_ImpulsInit							:= bGImpulsInitSprache,
	bI_OhneImpulsgeber						:= FALSE,
	strIO_GHdshk							:= strGHdshk_Bahn032501,
	strIO_GHdshk_Vorg						:= strGHdshk_Bahn031401,
	strIO_GHdshk_Nachf						:= strGHdshk_Bahn030601,
	strIO_GLmHand							:= strGLmHand,
	strIO_TrE								:= GDat.TrE_Daten[TrEId_032501],
	strIO_Stoerungen						:= strGStoerungen[iEins_Id]);

fbG6UmrichterBahn032501(
	sI_NetIDMaster					:= P_Ueberwachung_EtherCat.sNetId,
	sI_PfadXML						:= sGG6XMLPfad,
	sI_PfadSonderDatensatz			:= '',
	sI_Name							:= '=W325.EA1+S1-TA1',
	uiI_DevID						:= uiIDevID,
	uiI_FxId						:= FxId_032501,
	uiI_ProId						:= P_Umrichter,
	diI_Statuswort					:= udiIW325TA1Statuswort,
	usiI_Umrichterstatus			:= usiIW325TA1UmrichterStatus,
	uiI_Datensatz					:= 1,
	iI_Istfrequenz					:= uiIW325TA1Istfrequenz,
	tI_ZeitBremse					:= t#500ms,
	rI_Beschleunigung				:= 0.1,
	rI_Verzoegerung					:= 0.1,
	rI_Sollgeschwindigkeit			:= ABS(strGHdshk_Bahn032501.lr_Bahnspeed_Vorgabe),
	rI_Maxgeschwindigkeit			:= strGHdshk_Bahn032501.str_BahnSpeed.rVmaxSpeed,
	bI_Aktiv						:= TRUE,
	bI_FehlerQuitt					:= strGLmHand.bI_QuittStoerung,
	bI_Testbetrieb					:= gxTestbetriebOhneMaschineAktiv,
	bI_StartUmrichter				:= gxSicherheitsBereichQuittiertC[giSicher_C2_1],
	bI_Reglerfreigabe				:= gxSicherheitsBereichVerzOKC[giSicher_C2_1],
	bI_DrehrichtungVor				:= strGHdshk_Bahn032501.b_BahnVor,
	bI_DrehrichtungZurueck			:= strGHdshk_Bahn032501.b_BahnZurueck,
	bI_EtherCATOK					:= P_Ueberwachung_EtherCat.xAlles_OK,
	bI_DrehInv						:= FALSE,
	uiQ_EtherCATAdresse			  	=> uiGEtherCATAdresse_KEB[FxId_032501],
	iQ_Sollwert						=> uiQW325TA1Sollw,
	lrQ_Istwert						=> strGHdshk_Bahn032501.lr_Bahnspeed_Ist,
	diQ_Control						=> udiQW325TA1Control,
	bQ_Betriebsbereit				=> ,
	bQ_BremseLoesen					=> ,
	bQ_FehlerKEBDatenDownload		=> ,
	bQ_FehlerKeinIMAUmrichter		=> ,
	bQ_FehlerXMLDatei				=> ,
	bQ_FehlerParaLesen				=> ,
	bQ_FehlerParaSchreiben			=> ,
	bQ_FehlerAdresseLesen			=> ,
	strQ_Umrichterstatus			=> );

Aufruf_DisplayKEB.arI_DisplayKEB[FxId_032501]:=
	fbG6UmrichterBahn032501.strQ_Umrichterstatus.sConverterState;

fbJobBahn032501(
	bI_MitPCJob							:= FALSE,
	bI_FreigabeJobErzeugenSPS_Vorg		:= TRUE,
	bI_FreigabeJobErzeugenSPS_Nachf		:= FALSE,
	bI_FreigabeResetJob					:= astrGButtonManTransporte[ID_Bahn032501].bSchalt,
	bI_FreigabeResetBahn				:= astrGButtonManTransporte[ID_Bahn032501].bSchalt,
	bI_FreigabeFuerJob					:= bFreigabeFuerJob_C2_1,
	bI_ZusatzFreigabe					:= TRUE,
	bI_FreigabeFuerBuchen				:= bFreigabeFuerBuchen_C2_1,
	bI_MitAufBahnBeiVonBahn				:= FALSE,
	bI_BilderSammeln					:= FALSE, 
	bI_Querfoerderer					:= FALSE,
	bI_FreigabeAnBahnanfang				:= FALSE,
	bI_FreigabeAnsBahnende				:= FALSE,
	bI_ScannenAktiv						:= FALSE,
	bI_Testbetrieb						:= gxTestbetriebOhneMaschineAktiv,
	bI_FehlerQuittScanner				:= FALSE,
	bI_BeiResetJoblisteLoeschen			:= NOT bG3TecIstLeitsystem,
	iI_MaxAnzahlJobs					:= 1,
	iI_MaxAnzahlNoRead					:= 1,
	uiI_ProId							:= P_BahnJob,
	diI_SperrenQuellBahnNrVonPortal		:= 0,
	diI_SperrenZielBahnNrVonPortal		:= 0,
	tI_BisScannerDatenDa				:= t#0s,
	tI_Systemzeit						:= P_SystemzeitAuswerten.tDatumZeit_PC,
	strIO_GHdshk						:= strGHdshk_Bahn032501,
	strIO_GHdshk_Vorg					:= strGHdshk_Bahn031401,
	strIO_GHdshk_Nachf					:= strGHdshk_Bahn030601,
	strIO_TrE							:= GDat.TrE_Daten[TrEId_032501],
	strIO_TrE_Vorg						:= GDat.TrE_Daten[TrEId_031401],
	strIO_TrE_Nachf						:= GDat.TrE_Daten[TrEId_030601],
	strIO_ArbTab_Job					:= GJobDat.ArbTab_Job[TrEId_032501],
	strIO_GLmHand						:= strGLmHand,
	fbIO_Scanner						:= fbScanner_Leer,
	bQ_GrundOK							=> ,
	bQ_ResetAktiv						=> ,
	bQ_ScannerHatNichtGelesen			=> ,);
END_ACTION

ACTION Up_25_Bahn_032401:
fbHardwareBahn032401(
	uiI_ProId								:= P_BahnHardware,
	uiI_TrEId								:= TrEId_032401,
	uiI_AxId								:= 0,
	uiI_FehlerId							:= 4850,
	sI_Bahnname								:= '03.24.01',
	bI_Hand									:= fbEins[iEins_Id].OsHandEin,
	bI_Automatik							:= fbEins[iEins_Id].OsAutomatikEin,
	bI_Testbetrieb							:= gxTestbetriebOhneMaschineAktiv,
	bI_SicherheitOK							:= gxSicherheitsBereichQuittiertC[giSicher_C2_1],
	bI_FreigabeAutomatik					:= TRUE,
	bI_FreigabeHandVorZurueck				:= astrGButtonManTransporte[ID_Bahn032401].bSchalt,
	bI_BahnDarfZurueckHand					:= TRUE,
	bI_FreigabeReset						:= astrGButtonManTransporte[ID_Bahn032401].bSchalt,
	bI_StoerungAntrieb						:= NOT fbG6UmrichterBahn032401.bQ_Betriebsbereit,
	bI_Anfang								:= NOT bIW324Transp1AnfSpur1
													OR NOT bIW324Transp1AnfSpur2,
	bI_BelegtKontrolle						:= FALSE,
	bI_Ende									:= NOT bIW325Transp1AnfSpur1
													OR NOT bIW325Transp1AnfSpur2,
	bI_VorZurueckInversHand					:= FALSE,
	bI_AbbruchPosi_AufBahn					:= FALSE,
	bI_AbbruchPosi_VonBahn					:= FALSE,
	bI_BahnenGrundSchnell					:= FALSE,
	bI_GrundZurueck							:= FALSE,
	bI_OhneSynchronVonBahn					:= FALSE,
	bI_NachlaufAmAnfangEnde					:= FALSE,
	bI_MitUeberwachungTeilNichtFreigegeben	:= FALSE,
	bI_ImpulsInit							:= bGImpulsInitSprache,
	bI_OhneImpulsgeber						:= FALSE,
	strIO_GHdshk							:= strGHdshk_Bahn032401,
	strIO_GHdshk_Vorg						:= strGHdshk_Bahn030301,
	strIO_GHdshk_Nachf						:= strGHdshk_Bahn032501,
	strIO_GLmHand							:= strGLmHand,
	strIO_TrE								:= GDat.TrE_Daten[TrEId_032401],
	strIO_Stoerungen						:= strGStoerungen[iEins_Id]);

fbG6UmrichterBahn032401(
	sI_NetIDMaster					:= P_Ueberwachung_EtherCat.sNetId,
	sI_PfadXML						:= sGG6XMLPfad,
	sI_PfadSonderDatensatz			:= '',
	sI_Name							:= '=W324.EA1+S1-TA1',
	uiI_DevID						:= uiIDevID,
	uiI_FxId						:= FxId_032401,
	uiI_ProId						:= P_Umrichter,
	diI_Statuswort					:= udiIW324TA1Statuswort,
	usiI_Umrichterstatus			:= usiIW324TA1UmrichterStatus,
	uiI_Datensatz					:= 1,
	iI_Istfrequenz					:= uiIW324TA1Istfrequenz,
	tI_ZeitBremse					:= t#500ms,
	rI_Beschleunigung				:= 0.1,
	rI_Verzoegerung					:= 0.1,
	rI_Sollgeschwindigkeit			:= ABS(strGHdshk_Bahn032401.lr_Bahnspeed_Vorgabe),
	rI_Maxgeschwindigkeit			:= strGHdshk_Bahn032401.str_BahnSpeed.rVmaxSpeed,
	bI_Aktiv						:= TRUE,
	bI_FehlerQuitt					:= strGLmHand.bI_QuittStoerung,
	bI_Testbetrieb					:= gxTestbetriebOhneMaschineAktiv,
	bI_StartUmrichter				:= gxSicherheitsBereichQuittiertC[giSicher_C2_1],
	bI_Reglerfreigabe				:= gxSicherheitsBereichVerzOKC[giSicher_C2_1],
	bI_DrehrichtungVor				:= strGHdshk_Bahn032401.b_BahnVor,
	bI_DrehrichtungZurueck			:= strGHdshk_Bahn032401.b_BahnZurueck,
	bI_EtherCATOK					:= P_Ueberwachung_EtherCat.xAlles_OK,
	bI_DrehInv						:= TRUE,
	uiQ_EtherCATAdresse			  	=> uiGEtherCATAdresse_KEB[FxId_032401],
	iQ_Sollwert						=> uiQW324TA1Sollw,
	lrQ_Istwert						=> strGHdshk_Bahn032401.lr_Bahnspeed_Ist,
	diQ_Control						=> udiQW324TA1Control,
	bQ_Betriebsbereit				=> ,
	bQ_BremseLoesen					=> ,
	bQ_FehlerKEBDatenDownload		=> ,
	bQ_FehlerKeinIMAUmrichter		=> ,
	bQ_FehlerXMLDatei				=> ,
	bQ_FehlerParaLesen				=> ,
	bQ_FehlerParaSchreiben			=> ,
	bQ_FehlerAdresseLesen			=> ,
	strQ_Umrichterstatus			=> );

Aufruf_DisplayKEB.arI_DisplayKEB[FxId_032401]:=
	fbG6UmrichterBahn032401.strQ_Umrichterstatus.sConverterState;

fbJobBahn032401(
	bI_MitPCJob							:= TRUE,
	bI_FreigabeJobErzeugenSPS_Vorg		:= FALSE,
	bI_FreigabeJobErzeugenSPS_Nachf		:= FALSE,
	bI_FreigabeResetJob					:= astrGButtonManTransporte[ID_Bahn032401].bSchalt,
	bI_FreigabeResetBahn				:= astrGButtonManTransporte[ID_Bahn032401].bSchalt,
	bI_FreigabeFuerJob					:= bFreigabeFuerJob_C2_1,
	bI_ZusatzFreigabe					:= bFreigabeJob_Wippe_030301 
												AND iWippe_030301_IstAufPos = 3,
	bI_FreigabeFuerBuchen				:= bFreigabeFuerBuchen_C2_1,
	bI_MitAufBahnBeiVonBahn				:= FALSE,
	bI_BilderSammeln					:= FALSE,
	bI_Querfoerderer					:= FALSE,
	bI_FreigabeAnBahnanfang				:= FALSE,
	bI_FreigabeAnsBahnende				:= FALSE,
	bI_ScannenAktiv						:= FALSE,
	bI_Testbetrieb						:= gxTestbetriebOhneMaschineAktiv,
	bI_FehlerQuittScanner				:= FALSE,
	bI_BeiResetJoblisteLoeschen			:= NOT bG3TecIstLeitsystem,
	iI_MaxAnzahlJobs					:= 1,
	iI_MaxAnzahlNoRead					:= 1,
	uiI_ProId							:= P_BahnJob,
	diI_SperrenQuellBahnNrVonPortal		:= 0,
	diI_SperrenZielBahnNrVonPortal		:= 0,
	tI_BisScannerDatenDa				:= t#0s,
	tI_Systemzeit						:= P_SystemzeitAuswerten.tDatumZeit_PC,
	strIO_GHdshk						:= strGHdshk_Bahn032401,
	strIO_GHdshk_Vorg					:= strGHdshk_Bahn030301,
	strIO_GHdshk_Nachf					:= strGHdshk_Bahn032501,
	strIO_TrE							:= GDat.TrE_Daten[TrEId_032401],
	strIO_TrE_Vorg						:= GDat.TrE_Daten[TrEId_030301],
	strIO_TrE_Nachf						:= GDat.TrE_Daten[TrEId_032501],
	strIO_ArbTab_Job					:= GJobDat.ArbTab_Job[TrEId_032401],
	strIO_GLmHand						:= strGLmHand,
	fbIO_Scanner						:= fbScanner_Leer,
	bQ_GrundOK							=> ,
	bQ_ResetAktiv						=> ,
	bQ_ScannerHatNichtGelesen			=> ,
	bQ_ScannerFalscherBarcode			=> ,
	bQ_ScannerMaxAnzahlNoRead			=> );
END_ACTION

ACTION Up_26_Bahn_031501:
fbHardwareBahn031501(
	uiI_ProId								:= P_BahnHardware,
	uiI_TrEId								:= TrEId_031501,
	uiI_AxId								:= 0,
	uiI_FehlerId							:= 4800,
	sI_Bahnname								:= '03.15.01',
	bI_Hand									:= fbEins[iEins_Id].OsHandEin,
	bI_Automatik							:= fbEins[iEins_Id].OsAutomatikEin,
	bI_Testbetrieb							:= gxTestbetriebOhneMaschineAktiv,
	bI_SicherheitOK							:= gxSicherheitsBereichQuittiertC[giSicher_C2_1],
	bI_FreigabeAutomatik					:= TRUE,
	bI_FreigabeHandVorZurueck				:= astrGButtonManTransporte[ID_Bahn031501].bSchalt,
	bI_BahnDarfZurueckHand					:= TRUE,
	bI_FreigabeReset						:= astrGButtonManTransporte[ID_Bahn031501].bSchalt,
	bI_StoerungAntrieb						:= NOT fbG6UmrichterBahn031501.bQ_Betriebsbereit,
	bI_Anfang								:= NOT bIW315Transp1AnfSpur1
													OR NOT bIW315Transp1AnfSpur2,
	bI_BelegtKontrolle						:= FALSE,
	bI_Ende									:= NOT bIW315Transp1EndSpur1
													OR NOT bIW315Transp1EndSpur2,
	bI_VorZurueckInversHand					:= FALSE,
	bI_AbbruchPosi_AufBahn					:= FALSE,
	bI_AbbruchPosi_VonBahn					:= FALSE,
	bI_BahnenGrundSchnell					:= FALSE,
	bI_GrundZurueck							:= FALSE,
	bI_OhneSynchronVonBahn					:= FALSE,
	bI_NachlaufAmAnfangEnde					:= FALSE,
	bI_MitUeberwachungTeilNichtFreigegeben	:= FALSE,
	bI_ImpulsInit							:= bGImpulsInitSprache,
	bI_OhneImpulsgeber						:= FALSE,
	strIO_GHdshk							:= strGHdshk_Bahn031501,
	strIO_GHdshk_Vorg						:= strGHdshk_Bahn031401,
	strIO_GHdshk_Nachf						:= strGHdshk_Bahn030601,
	strIO_GLmHand							:= strGLmHand,
	strIO_TrE								:= GDat.TrE_Daten[TrEId_031501],
	strIO_Stoerungen						:= strGStoerungen[iEins_Id]);

fbG6UmrichterBahn031501(
	sI_NetIDMaster					:= P_Ueberwachung_EtherCat.sNetId,
	sI_PfadXML						:= sGG6XMLPfad,
	sI_PfadSonderDatensatz			:= '',
	sI_Name							:= '=W315.EA1+S1-TA1',
	uiI_DevID						:= uiIDevID,
	uiI_FxId						:= FxId_031501,
	uiI_ProId						:= P_Umrichter,
	diI_Statuswort					:= udiIW315TA1Statuswort,
	usiI_Umrichterstatus			:= usiIW315TA1UmrichterStatus,
	uiI_Datensatz					:= 1,
	iI_Istfrequenz					:= uiIW315TA1Istfrequenz,
	tI_ZeitBremse					:= t#500ms,
	rI_Beschleunigung				:= 0.1,
	rI_Verzoegerung					:= 0.1,
	rI_Sollgeschwindigkeit			:= ABS(strGHdshk_Bahn031501.lr_Bahnspeed_Vorgabe),
	rI_Maxgeschwindigkeit			:= strGHdshk_Bahn031501.str_BahnSpeed.rVmaxSpeed,
	bI_Aktiv						:= TRUE,
	bI_FehlerQuitt					:= strGLmHand.bI_QuittStoerung,
	bI_Testbetrieb					:= gxTestbetriebOhneMaschineAktiv,
	bI_StartUmrichter				:= gxSicherheitsBereichQuittiertC[giSicher_C2_1],
	bI_Reglerfreigabe				:= gxSicherheitsBereichVerzOKC[giSicher_C2_1],
	bI_DrehrichtungVor				:= strGHdshk_Bahn031501.b_BahnVor,
	bI_DrehrichtungZurueck			:= strGHdshk_Bahn031501.b_BahnZurueck,
	bI_EtherCATOK					:= P_Ueberwachung_EtherCat.xAlles_OK,
	bI_DrehInv						:= false,
	uiQ_EtherCATAdresse			  	=> uiGEtherCATAdresse_KEB[FxId_031501],
	iQ_Sollwert						=> uiQW315TA1Sollw,
	lrQ_Istwert						=> strGHdshk_Bahn031501.lr_Bahnspeed_Ist,
	diQ_Control						=> udiQW315TA1Control,
	bQ_Betriebsbereit				=> ,
	bQ_BremseLoesen					=> ,
	bQ_FehlerKEBDatenDownload		=> ,
	bQ_FehlerKeinIMAUmrichter		=> ,
	bQ_FehlerXMLDatei				=> ,
	bQ_FehlerParaLesen				=> ,
	bQ_FehlerParaSchreiben			=> ,
	bQ_FehlerAdresseLesen			=> ,
	strQ_Umrichterstatus			=> );

Aufruf_DisplayKEB.arI_DisplayKEB[FxId_031501]:=
	fbG6UmrichterBahn031501.strQ_Umrichterstatus.sConverterState;

fbJobBahn031501(
	bI_MitPCJob							:= FALSE,
	bI_FreigabeJobErzeugenSPS_Vorg		:= TRUE,
	bI_FreigabeJobErzeugenSPS_Nachf		:= FALSE,
	bI_FreigabeResetJob					:= astrGButtonManTransporte[ID_Bahn031501].bSchalt,
	bI_FreigabeResetBahn				:= astrGButtonManTransporte[ID_Bahn031501].bSchalt,
	bI_FreigabeFuerJob					:= bFreigabeFuerJob_C2_1,
	bI_ZusatzFreigabe					:= TRUE,
	bI_FreigabeFuerBuchen				:= bFreigabeFuerBuchen_C2_1,
	bI_MitAufBahnBeiVonBahn				:= FALSE,
	bI_BilderSammeln					:= FALSE, 
	bI_Querfoerderer					:= FALSE,
	bI_FreigabeAnBahnanfang				:= FALSE,
	bI_FreigabeAnsBahnende				:= FALSE,
	bI_ScannenAktiv						:= FALSE,
	bI_Testbetrieb						:= gxTestbetriebOhneMaschineAktiv,
	bI_FehlerQuittScanner				:= FALSE,
	bI_BeiResetJoblisteLoeschen			:= NOT bG3TecIstLeitsystem,
	iI_MaxAnzahlJobs					:= 1,
	iI_MaxAnzahlNoRead					:= 1,
	uiI_ProId							:= P_BahnJob,
	diI_SperrenQuellBahnNrVonPortal		:= 0,
	diI_SperrenZielBahnNrVonPortal		:= 0,
	tI_BisScannerDatenDa				:= t#0s,
	tI_Systemzeit						:= P_SystemzeitAuswerten.tDatumZeit_PC,
	strIO_GHdshk						:= strGHdshk_Bahn031501,
	strIO_GHdshk_Vorg					:= strGHdshk_Bahn031401,
	strIO_GHdshk_Nachf					:= strGHdshk_Bahn030601,
	strIO_TrE							:= GDat.TrE_Daten[TrEId_031501],
	strIO_TrE_Vorg						:= GDat.TrE_Daten[TrEId_031401],
	strIO_TrE_Nachf						:= GDat.TrE_Daten[TrEId_030601],
	strIO_ArbTab_Job					:= GJobDat.ArbTab_Job[TrEId_031501],
	strIO_GLmHand						:= strGLmHand,
	fbIO_Scanner						:= fbScanner_Leer,
	bQ_GrundOK							=> ,
	bQ_ResetAktiv						=> ,
	bQ_ScannerHatNichtGelesen			=> ,);
END_ACTION

ACTION Up_27_Bahn_031401:
fbHardwareBahn031401(
	uiI_ProId								:= P_BahnHardware,
	uiI_TrEId								:= TrEId_031401,
	uiI_AxId								:= 0,
	uiI_FehlerId							:= 4750,
	sI_Bahnname								:= '03.14.01',
	bI_Hand									:= fbEins[iEins_Id].OsHandEin,
	bI_Automatik							:= fbEins[iEins_Id].OsAutomatikEin,
	bI_Testbetrieb							:= gxTestbetriebOhneMaschineAktiv,
	bI_SicherheitOK							:= gxSicherheitsBereichQuittiertC[giSicher_C2_1],
	bI_FreigabeAutomatik					:= TRUE,
	bI_FreigabeHandVorZurueck				:= astrGButtonManTransporte[ID_Bahn031401].bSchalt,
	bI_BahnDarfZurueckHand					:= TRUE,
	bI_FreigabeReset						:= astrGButtonManTransporte[ID_Bahn031401].bSchalt,
	bI_StoerungAntrieb						:= NOT fbG6UmrichterBahn031401.bQ_Betriebsbereit,
	bI_Anfang								:= NOT bIW314Transp1AnfSpur1
													OR NOT bIW314Transp1AnfSpur2,
	bI_BelegtKontrolle						:= FALSE,
	bI_Ende									:= NOT bIW315Transp1AnfSpur1
													OR NOT bIW315Transp1AnfSpur2,
	bI_VorZurueckInversHand					:= FALSE,
	bI_AbbruchPosi_AufBahn					:= FALSE,
	bI_AbbruchPosi_VonBahn					:= FALSE,
	bI_BahnenGrundSchnell					:= FALSE,
	bI_GrundZurueck							:= FALSE,
	bI_OhneSynchronVonBahn					:= FALSE,
	bI_NachlaufAmAnfangEnde					:= FALSE,
	bI_MitUeberwachungTeilNichtFreigegeben	:= FALSE,
	bI_ImpulsInit							:= bGImpulsInitSprache,
	bI_OhneImpulsgeber						:= FALSE,
	strIO_GHdshk							:= strGHdshk_Bahn031401,
	strIO_GHdshk_Vorg						:= strGHdshk_Bahn030301,
	strIO_GHdshk_Nachf						:= strGHdshk_Bahn031501,
	strIO_GLmHand							:= strGLmHand,
	strIO_TrE								:= GDat.TrE_Daten[TrEId_031401],
	strIO_Stoerungen						:= strGStoerungen[iEins_Id]);

fbG6UmrichterBahn031401(
	sI_NetIDMaster					:= P_Ueberwachung_EtherCat.sNetId,
	sI_PfadXML						:= sGG6XMLPfad,
	sI_PfadSonderDatensatz			:= '',
	sI_Name							:= '=W314.EA1+S1-TA1',
	uiI_DevID						:= uiIDevID,
	uiI_FxId						:= FxId_031401,
	uiI_ProId						:= P_Umrichter,
	diI_Statuswort					:= udiIW314TA1Statuswort,
	usiI_Umrichterstatus			:= usiIW314TA1UmrichterStatus,
	uiI_Datensatz					:= 1,
	iI_Istfrequenz					:= uiIW314TA1Istfrequenz,
	tI_ZeitBremse					:= t#500ms,
	rI_Beschleunigung				:= 0.1,
	rI_Verzoegerung					:= 0.1,
	rI_Sollgeschwindigkeit			:= ABS(strGHdshk_Bahn031401.lr_Bahnspeed_Vorgabe),
	rI_Maxgeschwindigkeit			:= strGHdshk_Bahn031401.str_BahnSpeed.rVmaxSpeed,
	bI_Aktiv						:= TRUE,
	bI_FehlerQuitt					:= strGLmHand.bI_QuittStoerung,
	bI_Testbetrieb					:= gxTestbetriebOhneMaschineAktiv,
	bI_StartUmrichter				:= gxSicherheitsBereichQuittiertC[giSicher_C2_1],
	bI_Reglerfreigabe				:= gxSicherheitsBereichVerzOKC[giSicher_C2_1],
	bI_DrehrichtungVor				:= strGHdshk_Bahn031401.b_BahnVor,
	bI_DrehrichtungZurueck			:= strGHdshk_Bahn031401.b_BahnZurueck,
	bI_EtherCATOK					:= P_Ueberwachung_EtherCat.xAlles_OK,
	bI_DrehInv						:= TRUE,
	uiQ_EtherCATAdresse			  	=> uiGEtherCATAdresse_KEB[FxId_031401],
	iQ_Sollwert						=> uiQW314TA1Sollw,
	lrQ_Istwert						=> strGHdshk_Bahn031401.lr_Bahnspeed_Ist,
	diQ_Control						=> udiQW314TA1Control,
	bQ_Betriebsbereit				=> ,
	bQ_BremseLoesen					=> ,
	bQ_FehlerKEBDatenDownload		=> ,
	bQ_FehlerKeinIMAUmrichter		=> ,
	bQ_FehlerXMLDatei				=> ,
	bQ_FehlerParaLesen				=> ,
	bQ_FehlerParaSchreiben			=> ,
	bQ_FehlerAdresseLesen			=> ,
	strQ_Umrichterstatus			=> );

Aufruf_DisplayKEB.arI_DisplayKEB[FxId_031401]:=
	fbG6UmrichterBahn031401.strQ_Umrichterstatus.sConverterState;

fbJobBahn031401(
	bI_MitPCJob							:= TRUE,
	bI_FreigabeJobErzeugenSPS_Vorg		:= FALSE,
	bI_FreigabeJobErzeugenSPS_Nachf		:= FALSE,
	bI_FreigabeResetJob					:= astrGButtonManTransporte[ID_Bahn031401].bSchalt,
	bI_FreigabeResetBahn				:= astrGButtonManTransporte[ID_Bahn031401].bSchalt,
	bI_FreigabeFuerJob					:= bFreigabeFuerJob_C2_1,
	bI_ZusatzFreigabe					:= bFreigabeJob_Wippe_030301 
												AND iWippe_030301_IstAufPos = 2,
	bI_FreigabeFuerBuchen				:= bFreigabeFuerBuchen_C2_1,
	bI_MitAufBahnBeiVonBahn				:= FALSE,
	bI_BilderSammeln					:= FALSE,
	bI_Querfoerderer					:= FALSE,
	bI_FreigabeAnBahnanfang				:= FALSE,
	bI_FreigabeAnsBahnende				:= FALSE,
	bI_ScannenAktiv						:= FALSE,
	bI_Testbetrieb						:= gxTestbetriebOhneMaschineAktiv,
	bI_FehlerQuittScanner				:= FALSE,
	bI_BeiResetJoblisteLoeschen			:= NOT bG3TecIstLeitsystem,
	iI_MaxAnzahlJobs					:= 1,
	iI_MaxAnzahlNoRead					:= 1,
	uiI_ProId							:= P_BahnJob,
	diI_SperrenQuellBahnNrVonPortal		:= 0,
	diI_SperrenZielBahnNrVonPortal		:= 0,
	tI_BisScannerDatenDa				:= t#0s,
	tI_Systemzeit						:= P_SystemzeitAuswerten.tDatumZeit_PC,
	strIO_GHdshk						:= strGHdshk_Bahn031401,
	strIO_GHdshk_Vorg					:= strGHdshk_Bahn030301,
	strIO_GHdshk_Nachf					:= strGHdshk_Bahn031501,
	strIO_TrE							:= GDat.TrE_Daten[TrEId_031401],
	strIO_TrE_Vorg						:= GDat.TrE_Daten[TrEId_030301],
	strIO_TrE_Nachf						:= GDat.TrE_Daten[TrEId_031501],
	strIO_ArbTab_Job					:= GJobDat.ArbTab_Job[TrEId_031401],
	strIO_GLmHand						:= strGLmHand,
	fbIO_Scanner						:= fbScanner_Leer,
	bQ_GrundOK							=> ,
	bQ_ResetAktiv						=> ,
	bQ_ScannerHatNichtGelesen			=> ,
	bQ_ScannerFalscherBarcode			=> ,
	bQ_ScannerMaxAnzahlNoRead			=> );
END_ACTION

ACTION Up_28_Bahn_030501:
fbHardwareBahn030501(
	uiI_ProId								:= P_BahnHardware,
	uiI_TrEId								:= TrEId_030501,
	uiI_AxId								:= 0,
	uiI_FehlerId							:= 4400,
	sI_Bahnname								:= '03.05.01',
	bI_Hand									:= fbEins[iEins_Id].OsHandEin,
	bI_Automatik							:= fbEins[iEins_Id].OsAutomatikEin,
	bI_Testbetrieb							:= gxTestbetriebOhneMaschineAktiv,
	bI_SicherheitOK							:= gxSicherheitsBereichQuittiertC[giSicher_C2_1],
	bI_FreigabeAutomatik					:= TRUE,
	bI_FreigabeHandVorZurueck				:= astrGButtonManTransporte[ID_Bahn030501].bSchalt,
	bI_BahnDarfZurueckHand					:= TRUE,
	bI_FreigabeReset						:= astrGButtonManTransporte[ID_Bahn030501].bSchalt,
	bI_StoerungAntrieb						:= NOT fbG6UmrichterBahn030501.bQ_Betriebsbereit,
	bI_Anfang								:= NOT bIW305Transp1AnfSpur1
													OR NOT bIW305Transp1AnfSpur2,
	bI_BelegtKontrolle						:= FALSE,
	bI_Ende									:= NOT bIW305Transp1EndSpur1
													OR NOT bIW305Transp1EndSpur2,
	bI_VorZurueckInversHand					:= FALSE,
	bI_AbbruchPosi_AufBahn					:= FALSE,
	bI_AbbruchPosi_VonBahn					:= FALSE,
	bI_BahnenGrundSchnell					:= FALSE,
	bI_GrundZurueck							:= FALSE,
	bI_OhneSynchronVonBahn					:= FALSE,
	bI_NachlaufAmAnfangEnde					:= FALSE,
	bI_MitUeberwachungTeilNichtFreigegeben	:= FALSE,
	bI_ImpulsInit							:= bGImpulsInitSprache,
	bI_OhneImpulsgeber						:= FALSE,
	strIO_GHdshk							:= strGHdshk_Bahn030501,
	strIO_GHdshk_Vorg						:= strGHdshk_Bahn030401,
	strIO_GHdshk_Nachf						:= strGHdshk_Bahn030601,
	strIO_GLmHand							:= strGLmHand,
	strIO_TrE								:= GDat.TrE_Daten[TrEId_030501],
	strIO_Stoerungen						:= strGStoerungen[iEins_Id]);

fbG6UmrichterBahn030501(
	sI_NetIDMaster					:= P_Ueberwachung_EtherCat.sNetId,
	sI_PfadXML						:= sGG6XMLPfad,
	sI_PfadSonderDatensatz			:= '',
	sI_Name							:= '=W305.EA1+S1-TA1',
	uiI_DevID						:= uiIDevID,
	uiI_FxId						:= FxId_030501,
	uiI_ProId						:= P_Umrichter,
	diI_Statuswort					:= udiIW305TA1Statuswort,
	usiI_Umrichterstatus			:= usiIW305TA1UmrichterStatus,
	uiI_Datensatz					:= 1,
	iI_Istfrequenz					:= uiIW305TA1Istfrequenz,
	tI_ZeitBremse					:= t#500ms,
	rI_Beschleunigung				:= 0.1,
	rI_Verzoegerung					:= 0.1,
	rI_Sollgeschwindigkeit			:= ABS(strGHdshk_Bahn030501.lr_Bahnspeed_Vorgabe),
	rI_Maxgeschwindigkeit			:= strGHdshk_Bahn030501.str_BahnSpeed.rVmaxSpeed,
	bI_Aktiv						:= TRUE,
	bI_FehlerQuitt					:= strGLmHand.bI_QuittStoerung,
	bI_Testbetrieb					:= gxTestbetriebOhneMaschineAktiv,
	bI_StartUmrichter				:= gxSicherheitsBereichQuittiertC[giSicher_C2_1],
	bI_Reglerfreigabe				:= gxSicherheitsBereichVerzOKC[giSicher_C2_1],
	bI_DrehrichtungVor				:= strGHdshk_Bahn030501.b_BahnVor,
	bI_DrehrichtungZurueck			:= strGHdshk_Bahn030501.b_BahnZurueck,
	bI_EtherCATOK					:= P_Ueberwachung_EtherCat.xAlles_OK,
	bI_DrehInv						:= FALSE,
	uiQ_EtherCATAdresse			  	=> uiGEtherCATAdresse_KEB[FxId_030501],
	iQ_Sollwert						=> uiQW305TA1Sollw,
	lrQ_Istwert						=> strGHdshk_Bahn030501.lr_Bahnspeed_Ist,
	diQ_Control						=> udiQW305TA1Control,
	bQ_Betriebsbereit				=> ,
	bQ_BremseLoesen					=> ,
	bQ_FehlerKEBDatenDownload		=> ,
	bQ_FehlerKeinIMAUmrichter		=> ,
	bQ_FehlerXMLDatei				=> ,
	bQ_FehlerParaLesen				=> ,
	bQ_FehlerParaSchreiben			=> ,
	bQ_FehlerAdresseLesen			=> ,
	strQ_Umrichterstatus			=> );

Aufruf_DisplayKEB.arI_DisplayKEB[FxId_030501]:=
	fbG6UmrichterBahn030501.strQ_Umrichterstatus.sConverterState;

fbJobBahn030501(
	bI_MitPCJob							:= FALSE,
	bI_FreigabeJobErzeugenSPS_Vorg		:= TRUE,
	bI_FreigabeJobErzeugenSPS_Nachf		:= FALSE,
	bI_FreigabeResetJob					:= astrGButtonManTransporte[ID_Bahn030501].bSchalt,
	bI_FreigabeResetBahn				:= astrGButtonManTransporte[ID_Bahn030501].bSchalt,
	bI_FreigabeFuerJob					:= bFreigabeFuerJob_C2_1,
	bI_ZusatzFreigabe					:= TRUE,
	bI_FreigabeFuerBuchen				:= bFreigabeFuerBuchen_C2_1,
	bI_MitAufBahnBeiVonBahn				:= FALSE,
	bI_BilderSammeln					:= FALSE, 
	bI_Querfoerderer					:= FALSE,
	bI_FreigabeAnBahnanfang				:= FALSE,
	bI_FreigabeAnsBahnende				:= FALSE,
	bI_ScannenAktiv						:= FALSE,
	bI_Testbetrieb						:= gxTestbetriebOhneMaschineAktiv,
	bI_FehlerQuittScanner				:= FALSE,
	bI_BeiResetJoblisteLoeschen			:= NOT bG3TecIstLeitsystem,
	iI_MaxAnzahlJobs					:= 1,
	iI_MaxAnzahlNoRead					:= 1,
	uiI_ProId							:= P_BahnJob,
	diI_SperrenQuellBahnNrVonPortal		:= 0,
	diI_SperrenZielBahnNrVonPortal		:= 0,
	tI_BisScannerDatenDa				:= t#0s,
	tI_Systemzeit						:= P_SystemzeitAuswerten.tDatumZeit_PC,
	strIO_GHdshk						:= strGHdshk_Bahn030501,
	strIO_GHdshk_Vorg					:= strGHdshk_Bahn030401,
	strIO_GHdshk_Nachf					:= strGHdshk_Bahn030601,
	strIO_TrE							:= GDat.TrE_Daten[TrEId_030501],
	strIO_TrE_Vorg						:= GDat.TrE_Daten[TrEId_030401],
	strIO_TrE_Nachf						:= GDat.TrE_Daten[TrEId_030601],
	strIO_ArbTab_Job					:= GJobDat.ArbTab_Job[TrEId_030501],
	strIO_GLmHand						:= strGLmHand,
	fbIO_Scanner						:= fbScanner_Leer,
	bQ_GrundOK							=> ,
	bQ_ResetAktiv						=> ,
	bQ_ScannerHatNichtGelesen			=> ,
	bQ_ScannerFalscherBarcode			=> ,
	bQ_ScannerMaxAnzahlNoRead			=> );
END_ACTION

ACTION Up_29_Bahn_030401:
fbHardwareBahn030401(
	uiI_ProId								:= P_BahnHardware,
	uiI_TrEId								:= TrEId_030401,
	uiI_AxId								:= 0,
	uiI_FehlerId							:= 4350,
	sI_Bahnname								:= '03.04.01',
	bI_Hand									:= fbEins[iEins_Id].OsHandEin,
	bI_Automatik							:= fbEins[iEins_Id].OsAutomatikEin,
	bI_Testbetrieb							:= gxTestbetriebOhneMaschineAktiv,
	bI_SicherheitOK							:= gxSicherheitsBereichQuittiertC[giSicher_C2_1],
	bI_FreigabeAutomatik					:= TRUE,
	bI_FreigabeHandVorZurueck				:= astrGButtonManTransporte[ID_Bahn030401].bSchalt,
	bI_BahnDarfZurueckHand					:= TRUE,
	bI_FreigabeReset						:= astrGButtonManTransporte[ID_Bahn030401].bSchalt,
	bI_StoerungAntrieb						:= NOT fbG6UmrichterBahn030401.bQ_Betriebsbereit,
	bI_Anfang								:= NOT bIW304Transp1AnfSpur1
													OR NOT bIW304Transp1AnfSpur2,
	bI_BelegtKontrolle						:= FALSE,
	bI_Ende									:= NOT bIW305Transp1AnfSpur1
													OR NOT bIW305Transp1AnfSpur2,
	bI_VorZurueckInversHand					:= FALSE,
	bI_AbbruchPosi_AufBahn					:= FALSE,
	bI_AbbruchPosi_VonBahn					:= FALSE,
	bI_BahnenGrundSchnell					:= FALSE,
	bI_GrundZurueck							:= FALSE,
	bI_OhneSynchronVonBahn					:= FALSE,
	bI_NachlaufAmAnfangEnde					:= FALSE,
	bI_MitUeberwachungTeilNichtFreigegeben	:= FALSE,
	bI_ImpulsInit							:= bGImpulsInitSprache,
	bI_OhneImpulsgeber						:= FALSE,
	strIO_GHdshk							:= strGHdshk_Bahn030401,
	strIO_GHdshk_Vorg						:= strGHdshk_Bahn030301,
	strIO_GHdshk_Nachf						:= strGHdshk_Bahn030501,
	strIO_GLmHand							:= strGLmHand,
	strIO_TrE								:= GDat.TrE_Daten[TrEId_030401],
	strIO_Stoerungen						:= strGStoerungen[iEins_Id]);

fbG6UmrichterBahn030401(
	sI_NetIDMaster					:= P_Ueberwachung_EtherCat.sNetId,
	sI_PfadXML						:= sGG6XMLPfad,
	sI_PfadSonderDatensatz			:= '',
	sI_Name							:= '=W304.EA1+S1-TA1',
	uiI_DevID						:= uiIDevID,
	uiI_FxId						:= FxId_030401,
	uiI_ProId						:= P_Umrichter,
	diI_Statuswort					:= udiIW304TA1Statuswort,
	usiI_Umrichterstatus			:= usiIW304TA1UmrichterStatus,
	uiI_Datensatz					:= 1,
	iI_Istfrequenz					:= uiIW304TA1Istfrequenz,
	tI_ZeitBremse					:= t#500ms,
	rI_Beschleunigung				:= 0.1,
	rI_Verzoegerung					:= 0.1,
	rI_Sollgeschwindigkeit			:= ABS(strGHdshk_Bahn030401.lr_Bahnspeed_Vorgabe),
	rI_Maxgeschwindigkeit			:= strGHdshk_Bahn030401.str_BahnSpeed.rVmaxSpeed,
	bI_Aktiv						:= TRUE,
	bI_FehlerQuitt					:= strGLmHand.bI_QuittStoerung,
	bI_Testbetrieb					:= gxTestbetriebOhneMaschineAktiv,
	bI_StartUmrichter				:= gxSicherheitsBereichQuittiertC[giSicher_C2_1],
	bI_Reglerfreigabe				:= gxSicherheitsBereichVerzOKC[giSicher_C2_1],
	bI_DrehrichtungVor				:= strGHdshk_Bahn030401.b_BahnVor,
	bI_DrehrichtungZurueck			:= strGHdshk_Bahn030401.b_BahnZurueck,
	bI_EtherCATOK					:= P_Ueberwachung_EtherCat.xAlles_OK,
	bI_DrehInv						:= TRUE,
	uiQ_EtherCATAdresse			  	=> uiGEtherCATAdresse_KEB[FxId_030401],
	iQ_Sollwert						=> uiQW304TA1Sollw,
	lrQ_Istwert						=> strGHdshk_Bahn030401.lr_Bahnspeed_Ist,
	diQ_Control						=> udiQW304TA1Control,
	bQ_Betriebsbereit				=> ,
	bQ_BremseLoesen					=> ,
	bQ_FehlerKEBDatenDownload		=> ,
	bQ_FehlerKeinIMAUmrichter		=> ,
	bQ_FehlerXMLDatei				=> ,
	bQ_FehlerParaLesen				=> ,
	bQ_FehlerParaSchreiben			=> ,
	bQ_FehlerAdresseLesen			=> ,
	strQ_Umrichterstatus			=> );

Aufruf_DisplayKEB.arI_DisplayKEB[FxId_030401]:=
	fbG6UmrichterBahn030401.strQ_Umrichterstatus.sConverterState;

fbJobBahn030401(
	bI_MitPCJob							:= TRUE,
	bI_FreigabeJobErzeugenSPS_Vorg		:= FALSE,
	bI_FreigabeJobErzeugenSPS_Nachf		:= FALSE,
	bI_FreigabeResetJob					:= astrGButtonManTransporte[ID_Bahn030401].bSchalt,
	bI_FreigabeResetBahn				:= astrGButtonManTransporte[ID_Bahn030401].bSchalt,
	bI_FreigabeFuerJob					:= bFreigabeFuerJob_C2_1,
	bI_ZusatzFreigabe					:= bFreigabeJob_Wippe_030301 
												AND iWippe_030301_IstAufPos = 1,
	bI_FreigabeFuerBuchen				:= bFreigabeFuerBuchen_C2_1,
	bI_MitAufBahnBeiVonBahn				:= FALSE,
	bI_BilderSammeln					:= FALSE ,
	bI_Querfoerderer					:= FALSE,
	bI_FreigabeAnBahnanfang				:= FALSE,
	bI_FreigabeAnsBahnende				:= FALSE,
	bI_ScannenAktiv						:= FALSE,
	bI_Testbetrieb						:= gxTestbetriebOhneMaschineAktiv,
	bI_FehlerQuittScanner				:= FALSE,
	bI_BeiResetJoblisteLoeschen			:= NOT bG3TecIstLeitsystem,
	iI_MaxAnzahlJobs					:= 1,
	iI_MaxAnzahlNoRead					:= 1,
	uiI_ProId							:= P_BahnJob,
	diI_SperrenQuellBahnNrVonPortal		:= 0,
	diI_SperrenZielBahnNrVonPortal		:= 0,
	tI_BisScannerDatenDa				:= t#0s,
	tI_Systemzeit						:= P_SystemzeitAuswerten.tDatumZeit_PC,
	strIO_GHdshk						:= strGHdshk_Bahn030401,
	strIO_GHdshk_Vorg					:= strGHdshk_Bahn030301,
	strIO_GHdshk_Nachf					:= strGHdshk_Bahn030501,
	strIO_TrE							:= GDat.TrE_Daten[TrEId_030401],
	strIO_TrE_Vorg						:= GDat.TrE_Daten[TrEId_030301],
	strIO_TrE_Nachf						:= GDat.TrE_Daten[TrEId_030501],
	strIO_ArbTab_Job					:= GJobDat.ArbTab_Job[TrEId_030401],
	strIO_GLmHand						:= strGLmHand,
	fbIO_Scanner						:= fbScanner_Leer,
	bQ_GrundOK							=> ,
	bQ_ResetAktiv						=> ,
	bQ_ScannerHatNichtGelesen			=> ,
	bQ_ScannerFalscherBarcode			=> ,
	bQ_ScannerMaxAnzahlNoRead			=> );
END_ACTION

ACTION Up_30_Bahn_030301:

(*--------------------------*)
(* Sollposition Wippe       *)
(*--------------------------*)

IF	GDat.TrE_Daten[TrEId_030401].iJobStatus = iDatenAktiv
	AND	fbJobBahn030401.strBahnjob_Aktiv.diQuellId = strGHdshk_Bahn030301.di_PlatzId
	AND	GDat.TrE_Daten[TrEId_031401].iJobStatus = iSekNichtAktiv
	AND	GDat.TrE_Daten[TrEId_032401].iJobStatus = iSekNichtAktiv
THEN
	iWippe_030301_SollAufPos:= 1;

ELSIF GDat.TrE_Daten[TrEId_031401].iJobStatus = iDatenAktiv
	AND	fbJobBahn031401.strBahnjob_Aktiv.diQuellId = strGHdshk_Bahn030301.di_PlatzId
	AND	GDat.TrE_Daten[TrEId_030401].iJobStatus = iSekNichtAktiv
	AND	GDat.TrE_Daten[TrEId_032401].iJobStatus = iSekNichtAktiv
THEN
	iWippe_030301_SollAufPos:= 2;

ELSIF GDat.TrE_Daten[TrEId_032401].iJobStatus = iDatenAktiv
	AND	fbJobBahn032401.strBahnjob_Aktiv.diQuellId = strGHdshk_Bahn030301.di_PlatzId
	AND	GDat.TrE_Daten[TrEId_030401].iJobStatus = iSekNichtAktiv
	AND	GDat.TrE_Daten[TrEId_031401].iJobStatus = iSekNichtAktiv	
	OR ( GDat.TrE_Daten[TrEId_030301].iJobStatus = iDatenAktiv (* Darf Teile nur in Pos 3 Teile aufnehmen *)
		AND	( fbJobBahn030301.strBahnjob_Aktiv.diQuellId = strGHdshk_Bahn030201_Roll1.di_PlatzId
				OR fbJobBahn030301.strBahnjob_Aktiv.diQuellId = strGHdshk_Bahn030202_Roll2.di_PlatzId
				OR fbJobBahn030301.strBahnjob_Aktiv.diQuellId = strGHdshk_Bahn030205_Riem.di_PlatzId )
		AND GDat.TrE_Daten[TrEId_030301].iAnzahlPlatten = 0
		AND strGHdshk_Bahn030301.str_JobAktiv_VonBahn = eRolljobKeinJob )
THEN
	iWippe_030301_SollAufPos:= 3;

END_IF;

(*--------------------------*)
(* Zwischenmerker schreiben *)
(*--------------------------*)

IF	iWippe_030301_IstAufPos = 1
THEN
	strGHdshk_Zwischen_030301:= strGHdshk_Bahn030401;
	strTrEDaten_Zwischen_030301:= GDat.TrE_Daten[TrEId_030401];

ELSIF iWippe_030301_IstAufPos = 2
THEN
	strGHdshk_Zwischen_030301:= strGHdshk_Bahn031401;
	strTrEDaten_Zwischen_030301:= GDat.TrE_Daten[TrEId_031401];

ELSIF iWippe_030301_IstAufPos = 3
THEN
	strGHdshk_Zwischen_030301:= strGHdshk_Bahn032401;
	strTrEDaten_Zwischen_030301:= GDat.TrE_Daten[TrEId_032401];
ELSE
	strGHdshk_Zwischen_030301:= strBahnaustausch_Leer;
	strTrEDaten_Zwischen_030301:= TrE_Daten_Leer;
END_IF;


fbHardwareBahn030301(
	uiI_ProId								:= P_BahnHardware,
	uiI_TrEId								:= TrEId_030301,
	uiI_AxId								:= 0,
	uiI_FehlerId							:= 4300,
	sI_Bahnname								:= '03.03.01',
	bI_Hand									:= fbEins[iEins_Id].OsHandEin,
	bI_Automatik							:= fbEins[iEins_Id].OsAutomatikEin,
	bI_Testbetrieb							:= gxTestbetriebOhneMaschineAktiv,
	bI_SicherheitOK							:= gxSicherheitsBereichQuittiertC[giSicher_C2_1],
	bI_FreigabeAutomatik					:= TRUE,
	bI_FreigabeHandVorZurueck				:= astrGButtonManTransporte[ID_Bahn030301].bSchalt,
	bI_BahnDarfZurueckHand					:= TRUE,
	bI_FreigabeReset						:= astrGButtonManTransporte[ID_Bahn030301].bSchalt,
	bI_StoerungAntrieb						:= NOT fbG6UmrichterBahn030301.bQ_Betriebsbereit,
	bI_Anfang								:= NOT bIW303Transp1AnfSpur1
													OR NOT bIW303Transp1AnfSpur2,
	bI_BelegtKontrolle						:= FALSE,
	bI_Ende									:= NOT bIW303Transp1EndSpur1
													OR NOT bIW303Transp1EndSpur2,
	bI_VorZurueckInversHand					:= FALSE,
	bI_AbbruchPosi_AufBahn					:= FALSE,
	bI_AbbruchPosi_VonBahn					:= FALSE,
	bI_BahnenGrundSchnell					:= FALSE,
	bI_GrundZurueck							:= FALSE,
	bI_OhneSynchronVonBahn					:= FALSE ,	
	bI_NachlaufAmAnfangEnde					:= FALSE,
	bI_MitUeberwachungTeilNichtFreigegeben	:= FALSE,
	bI_ImpulsInit						:= bGImpulsInitSprache,
	bI_OhneImpulsgeber					:= FALSE,
	bI_AutoHandaufgabeAktiv				:= FALSE,
	bI_AutoHandentnahmeAktiv			:= FALSE,
	strIO_GHdshk						:= strGHdshk_Bahn030301,
	strIO_GHdshk_Vorg					:= strGHdshk_Bahn030205_Riem,
	strIO_GHdshk_Nachf					:= strGHdshk_Zwischen_030301,
	strIO_GLmHand						:= strGLmHand,
	strIO_TrE							:= GDat.TrE_Daten[TrEId_030301],
	strIO_Stoerungen					:= strGStoerungen[iEins_Id]);
	
fbG6UmrichterBahn030301(
	sI_NetIDMaster						:= P_Ueberwachung_EtherCat.sNetId,
	sI_PfadXML							:= sGG6XMLPfad,
	sI_PfadSonderDatensatz				:= '',
	sI_Name								:= '=W303.EA1+S1-TA1',
	uiI_FxId							:= FxId_030301,
	uiI_ProId							:= P_Umrichter,
	uiI_DevID							:= uiIDevID,
	diI_Statuswort						:= udiIW301TA1Statuswort,
	usiI_Umrichterstatus					:= usiIW303TA1UmrichterStatus,
	uiI_Datensatz						:= 1,
	iI_Istfrequenz						:= uiIW303TA1Istfrequenz,
	tI_ZeitBremse						:= t#500ms,
	rI_Beschleunigung						:= 0.1,
	rI_Verzoegerung						:= 0.1,
	rI_Sollgeschwindigkeit					:= LREAL_TO_REAL(ABS(strGHdshk_Bahn030301.lr_Bahnspeed_Vorgabe)),
	rI_Maxgeschwindigkeit					:= strGHdshk_Bahn030301.str_BahnSpeed.rVmaxSpeed,
	bI_Aktiv							:= TRUE,
	bI_FehlerQuitt						:= strGLmHand.bI_QuittStoerung,
	bI_Testbetrieb						:= gxTestbetriebOhneMaschineAktiv,
	bI_StartUmrichter						:= gxSicherheitsBereichQuittiertC[giSicher_C2_1],
	bI_Reglerfreigabe						:= gxSicherheitsBereichVerzOKC[giSicher_C2_1],
	bI_DrehrichtungVor					:= strGHdshk_Bahn030301.b_BahnVor,
	bI_DrehrichtungZurueck					:= strGHdshk_Bahn030301.b_BahnZurueck,
	bI_EtherCATOK						:= P_Ueberwachung_EtherCat.xAlles_OK,
	bI_DrehInv							:= FALSE,
	uiQ_EtherCATAdresse					=> uiGEtherCATAdresse_KEB[FxId_030301],
	iQ_Sollwert							=> uiQW303TA1Sollw,
	lrQ_Istwert							=> strGHdshk_Bahn030301.lr_Bahnspeed_Ist,
	diQ_Control							=> udiQW303TA1Control,
	bQ_Betriebsbereit						=> ,
	bQ_BremseLoesen						=> ,
	bQ_FehlerKEBDatenDownload				=> ,
	bQ_FehlerKeinIMAUmrichter				=> ,
	bQ_FehlerXMLDatei						=> ,
	bQ_FehlerParaLesen					=> ,
	bQ_FehlerParaSchreiben					=> ,
	bQ_FehlerAdresseLesen					=> ,
	strQ_Umrichterstatus					=> );

Aufruf_DisplayKEB.arI_DisplayKEB[FxId_030301]:=
	fbG6UmrichterBahn030301.strQ_Umrichterstatus.sConverterState;

(* Unklare Definition *)	
IF 	GJobDat.ArbTab_Job[TrEId_030301].JobZeile[1].diQuellId = strGHdshk_Bahn030202_Roll2.di_PlatzId
THEN 
	GJobDat.ArbTab_Job[TrEId_030301].JobZeile[1].diQuellId := strGHdshk_Bahn030201_Roll1.di_PlatzId;
END_IF

fbJobBahn030301(
	bI_MitPCJob								:= TRUE,
	bI_FreigabeJobErzeugenSPS_Vorg			:= FALSE,
	bI_FreigabeJobErzeugenSPS_Nachf			:= FALSE,
	bI_FreigabeResetJob						:= astrGButtonManTransporte[ID_Bahn030301].bSchalt,
	bI_FreigabeResetBahn					:= astrGButtonManTransporte[ID_Bahn030301].bSchalt,
	bI_FreigabeFuerJob						:= bFreigabeFuerJob_C2_1,
	bI_ZusatzFreigabe						:= strGHdshk_Anschlag030201.b_Grundstellung
												AND bFreigabeJob_Wippe_030301 
												AND iWippe_030301_IstAufPos = 3
												AND GJobDat.ArbTab_Job[TrEId_030301].JobZeile[1].diQuellId = strGHdshk_Bahn030201_Roll1.di_PlatzId,
	bI_FreigabeFuerBuchen					:= bFreigabeFuerBuchen_C2_1,
	bI_MitAufBahnBeiVonBahn					:= FALSE,
	bI_Querfoerderer						:= TRUE,
	bI_FreigabeAnBahnanfang					:= FALSE,
	bI_FreigabeAnsBahnende					:= FALSE,
	bI_BilderSammeln						:=  fbJobBahn030301.strBahnjob_Aktiv.aiPos_X[1] <= 1
												AND	fbJobBahn030301.strBahnjob_Aktiv.aiPos_X[2] <= 1
												AND	fbJobBahn030301.strBahnjob_Aktiv.aiPos_X[3] <= 1
												AND	fbJobBahn030301.strBahnjob_Aktiv.aiPos_X[4] <= 1
												AND	fbJobBahn030301.strBahnjob_Aktiv.arLaenge[1] <= strGHdshk_Bahn030301.str_Bahndaten.rRastermass_Laenge_LaengstePlatte
												AND	fbJobBahn030301.strBahnjob_Aktiv.arLaenge[2] <= strGHdshk_Bahn030301.str_Bahndaten.rRastermass_Laenge_LaengstePlatte ,
	bI_ScannenAktiv							:= FALSE,
	bI_Testbetrieb							:= gxTestbetriebOhneMaschineAktiv,
	bI_FehlerQuittScanner					:= FALSE,
	bI_BeiResetJoblisteLoeschen				:= NOT bG3TecIstLeitsystem,
	iI_MaxAnzahlJobs						:= 1,
	iI_MaxAnzahlNoRead						:= 1,
	uiI_ProId								:= P_BahnJob,
	diI_SperrenQuellBahnNrVonPortal			:= 0,
	diI_SperrenZielBahnNrVonPortal			:= 0,
	tI_BisScannerDatenDa					:= t#0s,
	tI_Systemzeit							:= P_SystemzeitAuswerten.tDatumZeit_PC,
	strIO_GHdshk							:= strGHdshk_Bahn030301,
	strIO_GHdshk_Vorg						:= strGHdshk_Bahn030205_Riem,
	strIO_GHdshk_Nachf						:= strGHdshk_Zwischen_030301,
	strIO_TrE								:= GDat.TrE_Daten[TrEId_030301],
	strIO_TrE_Vorg							:= GDat.TrE_Daten[TrEId_030202_Roll2],
	strIO_TrE_Nachf							:= strTrEDaten_Zwischen_030301,
	strIO_ArbTab_Job						:= GJobDat.ArbTab_Job[TrEId_030301],
	strIO_GLmHand							:= strGLmHand,
	fbIO_Scanner							:= fbScanner_Leer,
	bQ_GrundOK								=> ,
	bQ_ResetAktiv							=> ,
	bQ_ScannerHatNichtGelesen				=> ,
	bQ_ScannerFalscherBarcode				=> ,
	bQ_ScannerMaxAnzahlNoRead				=> );

	
	
(*---------------------------------*)
(* Zwischenmerker zurueckschreiben *)
(*---------------------------------*)

IF	iWippe_030301_IstAufPos = 1
THEN
	strGHdshk_Bahn030401:= strGHdshk_Zwischen_030301;
	GDat.TrE_Daten[TrEId_030401]:= strTrEDaten_Zwischen_030301;

ELSIF iWippe_030301_IstAufPos = 2
THEN
	strGHdshk_Bahn031401:= strGHdshk_Zwischen_030301;
	GDat.TrE_Daten[TrEId_031401]:= strTrEDaten_Zwischen_030301;

ELSIF iWippe_030301_IstAufPos = 3
THEN
	strGHdshk_Bahn032401:= strGHdshk_Zwischen_030301;
	GDat.TrE_Daten[TrEId_032401]:= strTrEDaten_Zwischen_030301;
END_IF;
END_ACTION

